Fanuc TP program (LS listing): kj_block_3.ls

/PROG  kj_block_3
/ATTR
COMMENT	= "19-04-11 14:31:32";
PROG_SIZE	= 0;
DEFAULT_GROUP	= 1, *, *, *, *;
/APPL
    ARC Welding Equipment: 1, *, *, *, *;
/MN
   1:  CALL HOME_ALL;
   1:  UFRAME_NUM = 1;
   1:  UTOOL_NUM = 3;
   1:  COL GUARD ADJUST 150;
   1:  MESSAGE[Teach Startpoint in PR90];
   1:  MESSAGE[Weld speed R100 in mm/sec];
   1:  MESSAGE[Retraction +Z in R101 in mm];
   1:  MESSAGE[Retraction speed in R102 in %];
   1:  !- Layer/Ebene 1;
   1:  PR[91] = PR[90];
   1:  PR[91,1] = PR[90,1] + 59.254;
   1:  PR[91,2] = PR[90,2] + 0.794;
   1:  PR[91,3] = PR[90,3] + 1.000;
   1:  PR[92] = PR[91];
   1:  PR[92,3] = PR[92,3] + R[101];
   1:J PR[92] R[102]% CNT100;
   1:L PR[91] 100mm/sec FINE RampTo R[100];
   1:  WAIT   2.00(sec);
   1:  CALL LASER_DRAHT_START;
   1:  PR[91,2] = PR[90,2] + 9.294;
   1:L PR[91] R[100]mm/sec CNT100;
   1:  PR[91,1] = PR[90,1] + 0.754;
   1:L PR[91] R[100]mm/sec CNT100;
   1:  PR[91,2] = PR[90,2] + 0.794;
   1:L PR[91] R[100]mm/sec CNT100;
   1:  PR[91,1] = PR[90,1] + 59.254;
   1:L PR[91] R[100]mm/sec CNT100TB   .50sec,CALL END_PUD;
   1:  WAIT    .50(sec);
   1:  DO[117:Laser Start]=OFF;
   1:  WAIT   10.00(sec);
   1:  PR[92] = PR[91];
   1:  PR[92,3] = PR[92,3] + R[101];
   1:J PR[92] R[102]% CNT100;
   1:  PR[91,1] = PR[90,1] + 56.803;
   1:  PR[91,2] = PR[90,2] + 2.144;
   1:  PR[92] = PR[91];
   1:  PR[92,3] = PR[92,3] + R[101];
   1:J PR[92] R[102]% CNT100;
   1:L PR[91] 100mm/sec FINE RampTo R[100];
   1:  WAIT   2.00(sec);
   1:  CALL LASER_DRAHT_START;
   1:  PR[91,1] = PR[90,1] + 57.904;
   1:  PR[91,2] = PR[90,2] + 3.246;
   1:L PR[91] R[100]mm/sec CNT100;
   1:  PR[91,2] = PR[90,2] + 5.367;
   1:L PR[91] R[100]mm/sec CNT100;
   1:  PR[91,1] = PR[90,1] + 54.681;
   1:  PR[91,2] = PR[90,2] + 2.144;
   1:L PR[91] R[100]mm/sec CNT100;
   1:  PR[91,1] = PR[90,1] + 52.560;
   1:L PR[91] R[100]mm/sec CNT100;
   1:  PR[91,1] = PR[90,1] + 57.904;
   1:  PR[91,2] = PR[90,2] + 7.489;
   1:L PR[91] R[100]mm/sec CNT100;
   1:  PR[91,2] = PR[90,2] + 7.944;
   1:L PR[91] R[100]mm/sec CNT100;
   1:  PR[91,1] = PR[90,1] + 56.239;
   1:L PR[91] R[100]mm/sec CNT100;
   1:  PR[91,1] = PR[90,1] + 50.439;
   1:  PR[91,2] = PR[90,2] + 2.144;
   1:L PR[91] R[100]mm/sec CNT100;
   1:  PR[91,1] = PR[90,1] + 48.317;
   1:L PR[91] R[100]mm/sec CNT100;
   1:  PR[91,1] = PR[90,1] + 54.117;
   1:  PR[91,2] = PR[90,2] + 7.944;
   1:L PR[91] R[100]mm/sec CNT100;
   1:  PR[91,1] = PR[90,1] + 51.996;
   1:L PR[91] R[100]mm/sec CNT100;
   1:  PR[91,1] = PR[90,1] + 46.196;
   1:  PR[91,2] = PR[90,2] + 2.144;
   1:L PR[91] R[100]mm/sec CNT100;
   1:  PR[91,1] = PR[90,1] + 44.075;
   1:L PR[91] R[100]mm/sec CNT100;
   1:  PR[91,1] = PR[90,1] + 49.875;
   1:  PR[91,2] = PR[90,2] + 7.944;
   1:L PR[91] R[100]mm/sec CNT100;
   1:  PR[91,1] = PR[90,1] + 47.753;
   1:L PR[91] R[100]mm/sec CNT100;
   1:  PR[91,1] = PR[90,1] + 41.953;
   1:  PR[91,2] = PR[90,2] + 2.144;
   1:L PR[91] R[100]mm/sec CNT100;
   1:  PR[91,1] = PR[90,1] + 39.832;
   1:L PR[91] R[100]mm/sec CNT100;
   1:  PR[91,1] = PR[90,1] + 45.632;
   1:  PR[91,2] = PR[90,2] + 7.944;
   1:L PR[91] R[100]mm/sec CNT100;
   1:  PR[91,1] = PR[90,1] + 43.511;
   1:L PR[91] R[100]mm/sec CNT100;
   1:  PR[91,1] = PR[90,1] + 37.711;
   1:  PR[91,2] = PR[90,2] + 2.144;
   1:L PR[91] R[100]mm/sec CNT100;
   1:  PR[91,1] = PR[90,1] + 35.589;
   1:L PR[91] R[100]mm/sec CNT100;
   1:  PR[91,1] = PR[90,1] + 41.389;
   1:  PR[91,2] = PR[90,2] + 7.944;
   1:L PR[91] R[100]mm/sec CNT100;
   1:  PR[91,1] = PR[90,1] + 39.268;
   1:L PR[91] R[100]mm/sec CNT100;
   1:  PR[91,1] = PR[90,1] + 33.468;
   1:  PR[91,2] = PR[90,2] + 2.144;
   1:L PR[91] R[100]mm/sec CNT100;
   1:  PR[91,1] = PR[90,1] + 31.347;
   1:L PR[91] R[100]mm/sec CNT100;
   1:  PR[91,1] = PR[90,1] + 37.147;
   1:  PR[91,2] = PR[90,2] + 7.944;
   1:L PR[91] R[100]mm/sec CNT100;
   1:  PR[91,1] = PR[90,1] + 35.025;
   1:L PR[91] R[100]mm/sec CNT100;
   1:  PR[91,1] = PR[90,1] + 29.225;
   1:  PR[91,2] = PR[90,2] + 2.144;
   1:L PR[91] R[100]mm/sec CNT100;
   1:  PR[91,1] = PR[90,1] + 27.104;
   1:L PR[91] R[100]mm/sec CNT100;
   1:  PR[91,1] = PR[90,1] + 32.904;
   1:  PR[91,2] = PR[90,2] + 7.944;
   1:L PR[91] R[100]mm/sec CNT100;
   1:  PR[91,1] = PR[90,1] + 30.783;
   1:L PR[91] R[100]mm/sec CNT100;
   1:  PR[91,1] = PR[90,1] + 24.983;
   1:  PR[91,2] = PR[90,2] + 2.144;
   1:L PR[91] R[100]mm/sec CNT100;
   1:  PR[91,1] = PR[90,1] + 22.862;
   1:L PR[91] R[100]mm/sec CNT100;
   1:  PR[91,1] = PR[90,1] + 28.662;
   1:  PR[91,2] = PR[90,2] + 7.944;
   1:L PR[91] R[100]mm/sec CNT100;
   1:  PR[91,1] = PR[90,1] + 26.540;
   1:L PR[91] R[100]mm/sec CNT100;
   1:  PR[91,1] = PR[90,1] + 20.740;
   1:  PR[91,2] = PR[90,2] + 2.144;
   1:L PR[91] R[100]mm/sec CNT100;
   1:  PR[91,1] = PR[90,1] + 18.619;
   1:L PR[91] R[100]mm/sec CNT100;
   1:  PR[91,1] = PR[90,1] + 24.419;
   1:  PR[91,2] = PR[90,2] + 7.944;
   1:L PR[91] R[100]mm/sec CNT100;
   1:  PR[91,1] = PR[90,1] + 22.298;
   1:L PR[91] R[100]mm/sec CNT100;
   1:  PR[91,1] = PR[90,1] + 16.498;
   1:  PR[91,2] = PR[90,2] + 2.144;
   1:L PR[91] R[100]mm/sec CNT100;
   1:  PR[91,1] = PR[90,1] + 14.376;
   1:L PR[91] R[100]mm/sec CNT100;
   1:  PR[91,1] = PR[90,1] + 20.176;
   1:  PR[91,2] = PR[90,2] + 7.944;
   1:L PR[91] R[100]mm/sec CNT100;
   1:  PR[91,1] = PR[90,1] + 18.055;
   1:L PR[91] R[100]mm/sec CNT100;
   1:  PR[91,1] = PR[90,1] + 12.255;
   1:  PR[91,2] = PR[90,2] + 2.144;
   1:L PR[91] R[100]mm/sec CNT100;
   1:  PR[91,1] = PR[90,1] + 10.134;
   1:L PR[91] R[100]mm/sec CNT100;
   1:  PR[91,1] = PR[90,1] + 15.934;
   1:  PR[91,2] = PR[90,2] + 7.944;
   1:L PR[91] R[100]mm/sec CNT100;
   1:  PR[91,1] = PR[90,1] + 13.812;
   1:L PR[91] R[100]mm/sec CNT100;
   1:  PR[91,1] = PR[90,1] + 8.012;
   1:  PR[91,2] = PR[90,2] + 2.144;
   1:L PR[91] R[100]mm/sec CNT100;
   1:  PR[91,1] = PR[90,1] + 5.891;
   1:L PR[91] R[100]mm/sec CNT100;
   1:  PR[91,1] = PR[90,1] + 11.691;
   1:  PR[91,2] = PR[90,2] + 7.944;
   1:L PR[91] R[100]mm/sec CNT100;
   1:  PR[91,1] = PR[90,1] + 9.570;
   1:L PR[91] R[100]mm/sec CNT100;
   1:  PR[91,1] = PR[90,1] + 3.770;
   1:  PR[91,2] = PR[90,2] + 2.144;
   1:L PR[91] R[100]mm/sec CNT100;
   1:  PR[91,1] = PR[90,1] + 2.104;
   1:L PR[91] R[100]mm/sec CNT100;
   1:  PR[91,2] = PR[90,2] + 2.600;
   1:L PR[91] R[100]mm/sec CNT100;
   1:  PR[91,1] = PR[90,1] + 7.448;
   1:  PR[91,2] = PR[90,2] + 7.944;
   1:L PR[91] R[100]mm/sec CNT100;
   1:  PR[91,1] = PR[90,1] + 5.327;
   1:L PR[91] R[100]mm/sec CNT100;
   1:  PR[91,1] = PR[90,1] + 2.104;
   1:  PR[91,2] = PR[90,2] + 4.722;
   1:L PR[91] R[100]mm/sec CNT100;
   1:  PR[91,2] = PR[90,2] + 6.843;
   1:L PR[91] R[100]mm/sec CNT100;
   1:  PR[91,1] = PR[90,1] + 3.206;
   1:  PR[91,2] = PR[90,2] + 7.944;
   1:L PR[91] R[100]mm/sec CNT100TB   .50sec,CALL END_PUD;
   1:  WAIT    .50(sec);
   1:  DO[117:Laser Start]=OFF;
   1:  WAIT   10.00(sec);
   1:  PR[92] = PR[91];
   1:  PR[92,3] = PR[92,3] + R[101];
   1:J PR[92] R[102]% CNT100;
   1:  !- Layer/Ebene 2;
   1:  PR[91] = PR[90];
   1:  PR[91,1] = PR[90,1] + 59.254;
   1:  PR[91,2] = PR[90,2] + 9.294;
   1:  PR[91,3] = PR[90,3] + 2.000;
   1:  PR[92] = PR[91];
   1:  PR[92,3] = PR[92,3] + R[101];
   1:J PR[92] R[102]% CNT100;
   1:L PR[91] 100mm/sec FINE RampTo R[100];
   1:  WAIT   2.00(sec);
   1:  CALL LASER_DRAHT_START;
   1:  PR[91,1] = PR[90,1] + 0.754;
   1:L PR[91] R[100]mm/sec CNT100;
   1:  PR[91,2] = PR[90,2] + 0.794;
   1:L PR[91] R[100]mm/sec CNT100;
   1:  PR[91,1] = PR[90,1] + 59.254;
   1:L PR[91] R[100]mm/sec CNT100;
   1:  PR[91,2] = PR[90,2] + 9.294;
   1:L PR[91] R[100]mm/sec CNT100TB   .50sec,CALL END_PUD;
   1:  WAIT    .50(sec);
   1:  DO[117:Laser Start]=OFF;
   1:  WAIT   10.00(sec);
   1:  PR[92] = PR[91];
   1:  PR[92,3] = PR[92,3] + R[101];
   1:J PR[92] R[102]% CNT100;
   1:  PR[91,1] = PR[90,1] + 57.904;
   1:  PR[91,2] = PR[90,2] + 6.843;
   1:  PR[92] = PR[91];
   1:  PR[92,3] = PR[92,3] + R[101];
   1:J PR[92] R[102]% CNT100;
   1:L PR[91] 100mm/sec FINE RampTo R[100];
   1:  WAIT   2.00(sec);
   1:  CALL LASER_DRAHT_START;
   1:  PR[91,1] = PR[90,1] + 56.803;
   1:  PR[91,2] = PR[90,2] + 7.944;
   1:L PR[91] R[100]mm/sec CNT100;
   1:  PR[91,1] = PR[90,1] + 54.681;
   1:L PR[91] R[100]mm/sec CNT100;
   1:  PR[91,1] = PR[90,1] + 57.904;
   1:  PR[91,2] = PR[90,2] + 4.722;
   1:L PR[91] R[100]mm/sec CNT100;
   1:  PR[91,2] = PR[90,2] + 2.600;
   1:L PR[91] R[100]mm/sec CNT100;
   1:  PR[91,1] = PR[90,1] + 52.560;
   1:  PR[91,2] = PR[90,2] + 7.944;
   1:L PR[91] R[100]mm/sec CNT100;
   1:  PR[91,1] = PR[90,1] + 50.439;
   1:L PR[91] R[100]mm/sec CNT100;
   1:  PR[91,1] = PR[90,1] + 56.239;
   1:  PR[91,2] = PR[90,2] + 2.144;
   1:L PR[91] R[100]mm/sec CNT100;
   1:  PR[91,1] = PR[90,1] + 54.117;
   1:L PR[91] R[100]mm/sec CNT100;
   1:  PR[91,1] = PR[90,1] + 48.317;
   1:  PR[91,2] = PR[90,2] + 7.944;
   1:L PR[91] R[100]mm/sec CNT100;
   1:  PR[91,1] = PR[90,1] + 46.196;
   1:L PR[91] R[100]mm/sec CNT100;
   1:  PR[91,1] = PR[90,1] + 51.996;
   1:  PR[91,2] = PR[90,2] + 2.144;
   1:L PR[91] R[100]mm/sec CNT100;
   1:  PR[91,1] = PR[90,1] + 49.875;
   1:L PR[91] R[100]mm/sec CNT100;
   1:  PR[91,1] = PR[90,1] + 44.075;
   1:  PR[91,2] = PR[90,2] + 7.944;
   1:L PR[91] R[100]mm/sec CNT100;
   1:  PR[91,1] = PR[90,1] + 41.953;
   1:L PR[91] R[100]mm/sec CNT100;
   1:  PR[91,1] = PR[90,1] + 47.753;
   1:  PR[91,2] = PR[90,2] + 2.144;
   1:L PR[91] R[100]mm/sec CNT100;
   1:  PR[91,1] = PR[90,1] + 45.632;
   1:L PR[91] R[100]mm/sec CNT100;
   1:  PR[91,1] = PR[90,1] + 39.832;
   1:  PR[91,2] = PR[90,2] + 7.944;
   1:L PR[91] R[100]mm/sec CNT100;
   1:  PR[91,1] = PR[90,1] + 37.711;
   1:L PR[91] R[100]mm/sec CNT100;
   1:  PR[91,1] = PR[90,1] + 43.511;
   1:  PR[91,2] = PR[90,2] + 2.144;
   1:L PR[91] R[100]mm/sec CNT100;
   1:  PR[91,1] = PR[90,1] + 41.389;
   1:L PR[91] R[100]mm/sec CNT100;
   1:  PR[91,1] = PR[90,1] + 35.589;
   1:  PR[91,2] = PR[90,2] + 7.944;
   1:L PR[91] R[100]mm/sec CNT100;
   1:  PR[91,1] = PR[90,1] + 33.468;
   1:L PR[91] R[100]mm/sec CNT100;
   1:  PR[91,1] = PR[90,1] + 39.268;
   1:  PR[91,2] = PR[90,2] + 2.144;
   1:L PR[91] R[100]mm/sec CNT100;
   1:  PR[91,1] = PR[90,1] + 37.147;
   1:L PR[91] R[100]mm/sec CNT100;
   1:  PR[91,1] = PR[90,1] + 31.347;
   1:  PR[91,2] = PR[90,2] + 7.944;
   1:L PR[91] R[100]mm/sec CNT100;
   1:  PR[91,1] = PR[90,1] + 29.226;
   1:L PR[91] R[100]mm/sec CNT100;
   1:  PR[91,1] = PR[90,1] + 35.026;
   1:  PR[91,2] = PR[90,2] + 2.144;
   1:L PR[91] R[100]mm/sec CNT100;
   1:  PR[91,1] = PR[90,1] + 32.904;
   1:L PR[91] R[100]mm/sec CNT100;
   1:  PR[91,1] = PR[90,1] + 27.104;
   1:  PR[91,2] = PR[90,2] + 7.944;
   1:L PR[91] R[100]mm/sec CNT100;
   1:  PR[91,1] = PR[90,1] + 24.983;
   1:L PR[91] R[100]mm/sec CNT100;
   1:  PR[91,1] = PR[90,1] + 30.783;
   1:  PR[91,2] = PR[90,2] + 2.144;
   1:L PR[91] R[100]mm/sec CNT100;
   1:  PR[91,1] = PR[90,1] + 28.662;
   1:L PR[91] R[100]mm/sec CNT100;
   1:  PR[91,1] = PR[90,1] + 22.862;
   1:  PR[91,2] = PR[90,2] + 7.944;
   1:L PR[91] R[100]mm/sec CNT100;
   1:  PR[91,1] = PR[90,1] + 20.740;
   1:L PR[91] R[100]mm/sec CNT100;
   1:  PR[91,1] = PR[90,1] + 26.540;
   1:  PR[91,2] = PR[90,2] + 2.144;
   1:L PR[91] R[100]mm/sec CNT100;
   1:  PR[91,1] = PR[90,1] + 24.419;
   1:L PR[91] R[100]mm/sec CNT100;
   1:  PR[91,1] = PR[90,1] + 18.619;
   1:  PR[91,2] = PR[90,2] + 7.944;
   1:L PR[91] R[100]mm/sec CNT100;
   1:  PR[91,1] = PR[90,1] + 16.498;
   1:L PR[91] R[100]mm/sec CNT100;
   1:  PR[91,1] = PR[90,1] + 22.298;
   1:  PR[91,2] = PR[90,2] + 2.144;
   1:L PR[91] R[100]mm/sec CNT100;
   1:  PR[91,1] = PR[90,1] + 20.176;
   1:L PR[91] R[100]mm/sec CNT100;
   1:  PR[91,1] = PR[90,1] + 14.376;
   1:  PR[91,2] = PR[90,2] + 7.944;
   1:L PR[91] R[100]mm/sec CNT100;
   1:  PR[91,1] = PR[90,1] + 12.255;
   1:L PR[91] R[100]mm/sec CNT100;
   1:  PR[91,1] = PR[90,1] + 18.055;
   1:  PR[91,2] = PR[90,2] + 2.144;
   1:L PR[91] R[100]mm/sec CNT100;
   1:  PR[91,1] = PR[90,1] + 15.934;
   1:L PR[91] R[100]mm/sec CNT100;
   1:  PR[91,1] = PR[90,1] + 10.134;
   1:  PR[91,2] = PR[90,2] + 7.944;
   1:L PR[91] R[100]mm/sec CNT100;
   1:  PR[91,1] = PR[90,1] + 8.012;
   1:L PR[91] R[100]mm/sec CNT100;
   1:  PR[91,1] = PR[90,1] + 13.812;
   1:  PR[91,2] = PR[90,2] + 2.144;
   1:L PR[91] R[100]mm/sec CNT100;
   1:  PR[91,1] = PR[90,1] + 11.691;
   1:L PR[91] R[100]mm/sec CNT100;
   1:  PR[91,1] = PR[90,1] + 5.891;
   1:  PR[91,2] = PR[90,2] + 7.944;
   1:L PR[91] R[100]mm/sec CNT100;
   1:  PR[91,1] = PR[90,1] + 3.770;
   1:L PR[91] R[100]mm/sec CNT100;
   1:  PR[91,1] = PR[90,1] + 9.570;
   1:  PR[91,2] = PR[90,2] + 2.144;
   1:L PR[91] R[100]mm/sec CNT100;
   1:  PR[91,1] = PR[90,1] + 7.448;
   1:L PR[91] R[100]mm/sec CNT100;
   1:  PR[91,1] = PR[90,1] + 2.104;
   1:  PR[91,2] = PR[90,2] + 7.489;
   1:L PR[91] R[100]mm/sec CNT100;
   1:  PR[91,2] = PR[90,2] + 5.367;
   1:L PR[91] R[100]mm/sec CNT100;
   1:  PR[91,1] = PR[90,1] + 5.327;
   1:  PR[91,2] = PR[90,2] + 2.144;
   1:L PR[91] R[100]mm/sec CNT100;
   1:  PR[91,1] = PR[90,1] + 3.206;
   1:L PR[91] R[100]mm/sec CNT100;
   1:  PR[91,1] = PR[90,1] + 2.104;
   1:  PR[91,2] = PR[90,2] + 3.246;
   1:L PR[91] R[100]mm/sec CNT100TB   .50sec,CALL END_PUD;
   1:  WAIT    .50(sec);
   1:  DO[117:Laser Start]=OFF;
   1:  WAIT   10.00(sec);
   1:  PR[92] = PR[91];
   1:  PR[92,3] = PR[92,3] + R[101];
   1:J PR[92] R[102]% CNT100;
   1:  !- Layer/Ebene 3;
   1:  PR[91] = PR[90];
   1:  PR[91,1] = PR[90,1] + 59.254;
   1:  PR[91,2] = PR[90,2] + 9.294;
   1:  PR[91,3] = PR[90,3] + 3.000;
   1:  PR[92] = PR[91];
   1:  PR[92,3] = PR[92,3] + R[101];
   1:J PR[92] R[102]% CNT100;
   1:L PR[91] 100mm/sec FINE RampTo R[100];
   1:  WAIT   2.00(sec);
   1:  CALL LASER_DRAHT_START;
   1:  PR[91,1] = PR[90,1] + 0.754;
   1:L PR[91] R[100]mm/sec CNT100;
   1:  PR[91,2] = PR[90,2] + 0.794;
   1:L PR[91] R[100]mm/sec CNT100;
   1:  PR[91,1] = PR[90,1] + 59.254;
   1:L PR[91] R[100]mm/sec CNT100;
   1:  PR[91,2] = PR[90,2] + 9.294;
   1:L PR[91] R[100]mm/sec CNT100TB   .50sec,CALL END_PUD;
   1:  WAIT    .50(sec);
   1:  DO[117:Laser Start]=OFF;
   1:  WAIT   10.00(sec);
   1:  PR[92] = PR[91];
   1:  PR[92,3] = PR[92,3] + R[101];
   1:J PR[92] R[102]% CNT100;
   1:  PR[91,1] = PR[90,1] + 56.803;
   1:  PR[91,2] = PR[90,2] + 2.144;
   1:  PR[92] = PR[91];
   1:  PR[92,3] = PR[92,3] + R[101];
   1:J PR[92] R[102]% CNT100;
   1:L PR[91] 100mm/sec FINE RampTo R[100];
   1:  WAIT   2.00(sec);
   1:  CALL LASER_DRAHT_START;
   1:  PR[91,1] = PR[90,1] + 57.904;
   1:  PR[91,2] = PR[90,2] + 3.246;
   1:L PR[91] R[100]mm/sec CNT100;
   1:  PR[91,2] = PR[90,2] + 5.367;
   1:L PR[91] R[100]mm/sec CNT100;
   1:  PR[91,1] = PR[90,1] + 54.681;
   1:  PR[91,2] = PR[90,2] + 2.144;
   1:L PR[91] R[100]mm/sec CNT100;
   1:  PR[91,1] = PR[90,1] + 52.560;
   1:L PR[91] R[100]mm/sec CNT100;
   1:  PR[91,1] = PR[90,1] + 57.904;
   1:  PR[91,2] = PR[90,2] + 7.489;
   1:L PR[91] R[100]mm/sec CNT100;
   1:  PR[91,2] = PR[90,2] + 7.944;
   1:L PR[91] R[100]mm/sec CNT100;
   1:  PR[91,1] = PR[90,1] + 56.239;
   1:L PR[91] R[100]mm/sec CNT100;
   1:  PR[91,1] = PR[90,1] + 50.439;
   1:  PR[91,2] = PR[90,2] + 2.144;
   1:L PR[91] R[100]mm/sec CNT100;
   1:  PR[91,1] = PR[90,1] + 48.317;
   1:L PR[91] R[100]mm/sec CNT100;
   1:  PR[91,1] = PR[90,1] + 54.117;
   1:  PR[91,2] = PR[90,2] + 7.944;
   1:L PR[91] R[100]mm/sec CNT100;
   1:  PR[91,1] = PR[90,1] + 51.996;
   1:L PR[91] R[100]mm/sec CNT100;
   1:  PR[91,1] = PR[90,1] + 46.196;
   1:  PR[91,2] = PR[90,2] + 2.144;
   1:L PR[91] R[100]mm/sec CNT100;
   1:  PR[91,1] = PR[90,1] + 44.075;
   1:L PR[91] R[100]mm/sec CNT100;
   1:  PR[91,1] = PR[90,1] + 49.875;
   1:  PR[91,2] = PR[90,2] + 7.944;
   1:L PR[91] R[100]mm/sec CNT100;
   1:  PR[91,1] = PR[90,1] + 47.753;
   1:L PR[91] R[100]mm/sec CNT100;
   1:  PR[91,1] = PR[90,1] + 41.953;
   1:  PR[91,2] = PR[90,2] + 2.144;
   1:L PR[91] R[100]mm/sec CNT100;
   1:  PR[91,1] = PR[90,1] + 39.832;
   1:L PR[91] R[100]mm/sec CNT100;
   1:  PR[91,1] = PR[90,1] + 45.632;
   1:  PR[91,2] = PR[90,2] + 7.944;
   1:L PR[91] R[100]mm/sec CNT100;
   1:  PR[91,1] = PR[90,1] + 43.511;
   1:L PR[91] R[100]mm/sec CNT100;
   1:  PR[91,1] = PR[90,1] + 37.711;
   1:  PR[91,2] = PR[90,2] + 2.144;
   1:L PR[91] R[100]mm/sec CNT100;
   1:  PR[91,1] = PR[90,1] + 35.589;
   1:L PR[91] R[100]mm/sec CNT100;
   1:  PR[91,1] = PR[90,1] + 41.389;
   1:  PR[91,2] = PR[90,2] + 7.944;
   1:L PR[91] R[100]mm/sec CNT100;
   1:  PR[91,1] = PR[90,1] + 39.268;
   1:L PR[91] R[100]mm/sec CNT100;
   1:  PR[91,1] = PR[90,1] + 33.468;
   1:  PR[91,2] = PR[90,2] + 2.144;
   1:L PR[91] R[100]mm/sec CNT100;
   1:  PR[91,1] = PR[90,1] + 31.347;
   1:L PR[91] R[100]mm/sec CNT100;
   1:  PR[91,1] = PR[90,1] + 37.147;
   1:  PR[91,2] = PR[90,2] + 7.944;
   1:L PR[91] R[100]mm/sec CNT100;
   1:  PR[91,1] = PR[90,1] + 35.025;
   1:L PR[91] R[100]mm/sec CNT100;
   1:  PR[91,1] = PR[90,1] + 29.225;
   1:  PR[91,2] = PR[90,2] + 2.144;
   1:L PR[91] R[100]mm/sec CNT100;
   1:  PR[91,1] = PR[90,1] + 27.104;
   1:L PR[91] R[100]mm/sec CNT100;
   1:  PR[91,1] = PR[90,1] + 32.904;
   1:  PR[91,2] = PR[90,2] + 7.944;
   1:L PR[91] R[100]mm/sec CNT100;
   1:  PR[91,1] = PR[90,1] + 30.783;
   1:L PR[91] R[100]mm/sec CNT100;
   1:  PR[91,1] = PR[90,1] + 24.983;
   1:  PR[91,2] = PR[90,2] + 2.144;
   1:L PR[91] R[100]mm/sec CNT100;
   1:  PR[91,1] = PR[90,1] + 22.862;
   1:L PR[91] R[100]mm/sec CNT100;
   1:  PR[91,1] = PR[90,1] + 28.662;
   1:  PR[91,2] = PR[90,2] + 7.944;
   1:L PR[91] R[100]mm/sec CNT100;
   1:  PR[91,1] = PR[90,1] + 26.540;
   1:L PR[91] R[100]mm/sec CNT100;
   1:  PR[91,1] = PR[90,1] + 20.740;
   1:  PR[91,2] = PR[90,2] + 2.144;
   1:L PR[91] R[100]mm/sec CNT100;
   1:  PR[91,1] = PR[90,1] + 18.619;
   1:L PR[91] R[100]mm/sec CNT100;
   1:  PR[91,1] = PR[90,1] + 24.419;
   1:  PR[91,2] = PR[90,2] + 7.944;
   1:L PR[91] R[100]mm/sec CNT100;
   1:  PR[91,1] = PR[90,1] + 22.298;
   1:L PR[91] R[100]mm/sec CNT100;
   1:  PR[91,1] = PR[90,1] + 16.498;
   1:  PR[91,2] = PR[90,2] + 2.144;
   1:L PR[91] R[100]mm/sec CNT100;
   1:  PR[91,1] = PR[90,1] + 14.376;
   1:L PR[91] R[100]mm/sec CNT100;
   1:  PR[91,1] = PR[90,1] + 20.176;
   1:  PR[91,2] = PR[90,2] + 7.944;
   1:L PR[91] R[100]mm/sec CNT100;
   1:  PR[91,1] = PR[90,1] + 18.055;
   1:L PR[91] R[100]mm/sec CNT100;
   1:  PR[91,1] = PR[90,1] + 12.255;
   1:  PR[91,2] = PR[90,2] + 2.144;
   1:L PR[91] R[100]mm/sec CNT100;
   1:  PR[91,1] = PR[90,1] + 10.134;
   1:L PR[91] R[100]mm/sec CNT100;
   1:  PR[91,1] = PR[90,1] + 15.934;
   1:  PR[91,2] = PR[90,2] + 7.944;
   1:L PR[91] R[100]mm/sec CNT100;
   1:  PR[91,1] = PR[90,1] + 13.812;
   1:L PR[91] R[100]mm/sec CNT100;
   1:  PR[91,1] = PR[90,1] + 8.012;
   1:  PR[91,2] = PR[90,2] + 2.144;
   1:L PR[91] R[100]mm/sec CNT100;
   1:  PR[91,1] = PR[90,1] + 5.891;
   1:L PR[91] R[100]mm/sec CNT100;
   1:  PR[91,1] = PR[90,1] + 11.691;
   1:  PR[91,2] = PR[90,2] + 7.944;
   1:L PR[91] R[100]mm/sec CNT100;
   1:  PR[91,1] = PR[90,1] + 9.570;
   1:L PR[91] R[100]mm/sec CNT100;
   1:  PR[91,1] = PR[90,1] + 3.770;
   1:  PR[91,2] = PR[90,2] + 2.144;
   1:L PR[91] R[100]mm/sec CNT100;
   1:  PR[91,1] = PR[90,1] + 2.104;
   1:L PR[91] R[100]mm/sec CNT100;
   1:  PR[91,2] = PR[90,2] + 2.600;
   1:L PR[91] R[100]mm/sec CNT100;
   1:  PR[91,1] = PR[90,1] + 7.448;
   1:  PR[91,2] = PR[90,2] + 7.944;
   1:L PR[91] R[100]mm/sec CNT100;
   1:  PR[91,1] = PR[90,1] + 5.327;
   1:L PR[91] R[100]mm/sec CNT100;
   1:  PR[91,1] = PR[90,1] + 2.104;
   1:  PR[91,2] = PR[90,2] + 4.722;
   1:L PR[91] R[100]mm/sec CNT100;
   1:  PR[91,2] = PR[90,2] + 6.843;
   1:L PR[91] R[100]mm/sec CNT100;
   1:  PR[91,1] = PR[90,1] + 3.206;
   1:  PR[91,2] = PR[90,2] + 7.944;
   1:L PR[91] R[100]mm/sec CNT100TB   .50sec,CALL END_PUD;
   1:  WAIT    .50(sec);
   1:  DO[117:Laser Start]=OFF;
   1:  WAIT   10.00(sec);
   1:  PR[92] = PR[91];
   1:  PR[92,3] = PR[92,3] + R[101];
   1:J PR[92] R[102]% CNT100;
   1:  !- Layer/Ebene 4;
   1:  PR[91] = PR[90];
   1:  PR[91,1] = PR[90,1] + 0.754;
   1:  PR[91,2] = PR[90,2] + 0.794;
   1:  PR[91,3] = PR[90,3] + 4.000;
   1:  PR[92] = PR[91];
   1:  PR[92,3] = PR[92,3] + R[101];
   1:J PR[92] R[102]% CNT100;
   1:L PR[91] 100mm/sec FINE RampTo R[100];
   1:  WAIT   2.00(sec);
   1:  CALL LASER_DRAHT_START;
   1:  PR[91,1] = PR[90,1] + 59.254;
   1:L PR[91] R[100]mm/sec CNT100;
   1:  PR[91,2] = PR[90,2] + 9.294;
   1:L PR[91] R[100]mm/sec CNT100;
   1:  PR[91,1] = PR[90,1] + 0.754;
   1:L PR[91] R[100]mm/sec CNT100;
   1:  PR[91,2] = PR[90,2] + 0.794;
   1:L PR[91] R[100]mm/sec CNT100TB   .50sec,CALL END_PUD;
   1:  WAIT    .50(sec);
   1:  DO[117:Laser Start]=OFF;
   1:  WAIT   10.00(sec);
   1:  PR[92] = PR[91];
   1:  PR[92,3] = PR[92,3] + R[101];
   1:J PR[92] R[102]% CNT100;
   1:  PR[91,1] = PR[90,1] + 2.104;
   1:  PR[91,2] = PR[90,2] + 3.246;
   1:  PR[92] = PR[91];
   1:  PR[92,3] = PR[92,3] + R[101];
   1:J PR[92] R[102]% CNT100;
   1:L PR[91] 100mm/sec FINE RampTo R[100];
   1:  WAIT   2.00(sec);
   1:  CALL LASER_DRAHT_START;
   1:  PR[91,1] = PR[90,1] + 3.206;
   1:  PR[91,2] = PR[90,2] + 2.144;
   1:L PR[91] R[100]mm/sec CNT100;
   1:  PR[91,1] = PR[90,1] + 5.327;
   1:L PR[91] R[100]mm/sec CNT100;
   1:  PR[91,1] = PR[90,1] + 2.104;
   1:  PR[91,2] = PR[90,2] + 5.367;
   1:L PR[91] R[100]mm/sec CNT100;
   1:  PR[91,2] = PR[90,2] + 7.489;
   1:L PR[91] R[100]mm/sec CNT100;
   1:  PR[91,1] = PR[90,1] + 7.448;
   1:  PR[91,2] = PR[90,2] + 2.144;
   1:L PR[91] R[100]mm/sec CNT100;
   1:  PR[91,1] = PR[90,1] + 9.570;
   1:L PR[91] R[100]mm/sec CNT100;
   1:  PR[91,1] = PR[90,1] + 3.770;
   1:  PR[91,2] = PR[90,2] + 7.944;
   1:L PR[91] R[100]mm/sec CNT100;
   1:  PR[91,1] = PR[90,1] + 5.891;
   1:L PR[91] R[100]mm/sec CNT100;
   1:  PR[91,1] = PR[90,1] + 11.691;
   1:  PR[91,2] = PR[90,2] + 2.144;
   1:L PR[91] R[100]mm/sec CNT100;
   1:  PR[91,1] = PR[90,1] + 13.812;
   1:L PR[91] R[100]mm/sec CNT100;
   1:  PR[91,1] = PR[90,1] + 8.012;
   1:  PR[91,2] = PR[90,2] + 7.944;
   1:L PR[91] R[100]mm/sec CNT100;
   1:  PR[91,1] = PR[90,1] + 10.134;
   1:L PR[91] R[100]mm/sec CNT100;
   1:  PR[91,1] = PR[90,1] + 15.934;
   1:  PR[91,2] = PR[90,2] + 2.144;
   1:L PR[91] R[100]mm/sec CNT100;
   1:  PR[91,1] = PR[90,1] + 18.055;
   1:L PR[91] R[100]mm/sec CNT100;
   1:  PR[91,1] = PR[90,1] + 12.255;
   1:  PR[91,2] = PR[90,2] + 7.944;
   1:L PR[91] R[100]mm/sec CNT100;
   1:  PR[91,1] = PR[90,1] + 14.376;
   1:L PR[91] R[100]mm/sec CNT100;
   1:  PR[91,1] = PR[90,1] + 20.176;
   1:  PR[91,2] = PR[90,2] + 2.144;
   1:L PR[91] R[100]mm/sec CNT100;
   1:  PR[91,1] = PR[90,1] + 22.298;
   1:L PR[91] R[100]mm/sec CNT100;
   1:  PR[91,1] = PR[90,1] + 16.498;
   1:  PR[91,2] = PR[90,2] + 7.944;
   1:L PR[91] R[100]mm/sec CNT100;
   1:  PR[91,1] = PR[90,1] + 18.619;
   1:L PR[91] R[100]mm/sec CNT100;
   1:  PR[91,1] = PR[90,1] + 24.419;
   1:  PR[91,2] = PR[90,2] + 2.144;
   1:L PR[91] R[100]mm/sec CNT100;
   1:  PR[91,1] = PR[90,1] + 26.540;
   1:L PR[91] R[100]mm/sec CNT100;
   1:  PR[91,1] = PR[90,1] + 20.740;
   1:  PR[91,2] = PR[90,2] + 7.944;
   1:L PR[91] R[100]mm/sec CNT100;
   1:  PR[91,1] = PR[90,1] + 22.862;
   1:L PR[91] R[100]mm/sec CNT100;
   1:  PR[91,1] = PR[90,1] + 28.662;
   1:  PR[91,2] = PR[90,2] + 2.144;
   1:L PR[91] R[100]mm/sec CNT100;
   1:  PR[91,1] = PR[90,1] + 30.783;
   1:L PR[91] R[100]mm/sec CNT100;
   1:  PR[91,1] = PR[90,1] + 24.983;
   1:  PR[91,2] = PR[90,2] + 7.944;
   1:L PR[91] R[100]mm/sec CNT100;
   1:  PR[91,1] = PR[90,1] + 27.104;
   1:L PR[91] R[100]mm/sec CNT100;
   1:  PR[91,1] = PR[90,1] + 32.904;
   1:  PR[91,2] = PR[90,2] + 2.144;
   1:L PR[91] R[100]mm/sec CNT100;
   1:  PR[91,1] = PR[90,1] + 35.026;
   1:L PR[91] R[100]mm/sec CNT100;
   1:  PR[91,1] = PR[90,1] + 29.226;
   1:  PR[91,2] = PR[90,2] + 7.944;
   1:L PR[91] R[100]mm/sec CNT100;
   1:  PR[91,1] = PR[90,1] + 31.347;
   1:L PR[91] R[100]mm/sec CNT100;
   1:  PR[91,1] = PR[90,1] + 37.147;
   1:  PR[91,2] = PR[90,2] + 2.144;
   1:L PR[91] R[100]mm/sec CNT100;
   1:  PR[91,1] = PR[90,1] + 39.268;
   1:L PR[91] R[100]mm/sec CNT100;
   1:  PR[91,1] = PR[90,1] + 33.468;
   1:  PR[91,2] = PR[90,2] + 7.944;
   1:L PR[91] R[100]mm/sec CNT100;
   1:  PR[91,1] = PR[90,1] + 35.589;
   1:L PR[91] R[100]mm/sec CNT100;
   1:  PR[91,1] = PR[90,1] + 41.389;
   1:  PR[91,2] = PR[90,2] + 2.144;
   1:L PR[91] R[100]mm/sec CNT100;
   1:  PR[91,1] = PR[90,1] + 43.511;
   1:L PR[91] R[100]mm/sec CNT100;
   1:  PR[91,1] = PR[90,1] + 37.711;
   1:  PR[91,2] = PR[90,2] + 7.944;
   1:L PR[91] R[100]mm/sec CNT100;
   1:  PR[91,1] = PR[90,1] + 39.832;
   1:L PR[91] R[100]mm/sec CNT100;
   1:  PR[91,1] = PR[90,1] + 45.632;
   1:  PR[91,2] = PR[90,2] + 2.144;
   1:L PR[91] R[100]mm/sec CNT100;
   1:  PR[91,1] = PR[90,1] + 47.753;
   1:L PR[91] R[100]mm/sec CNT100;
   1:  PR[91,1] = PR[90,1] + 41.953;
   1:  PR[91,2] = PR[90,2] + 7.944;
   1:L PR[91] R[100]mm/sec CNT100;
   1:  PR[91,1] = PR[90,1] + 44.075;
   1:L PR[91] R[100]mm/sec CNT100;
   1:  PR[91,1] = PR[90,1] + 49.875;
   1:  PR[91,2] = PR[90,2] + 2.144;
   1:L PR[91] R[100]mm/sec CNT100;
   1:  PR[91,1] = PR[90,1] + 51.996;
   1:L PR[91] R[100]mm/sec CNT100;
   1:  PR[91,1] = PR[90,1] + 46.196;
   1:  PR[91,2] = PR[90,2] + 7.944;
   1:L PR[91] R[100]mm/sec CNT100;
   1:  PR[91,1] = PR[90,1] + 48.317;
   1:L PR[91] R[100]mm/sec CNT100;
   1:  PR[91,1] = PR[90,1] + 54.117;
   1:  PR[91,2] = PR[90,2] + 2.144;
   1:L PR[91] R[100]mm/sec CNT100;
   1:  PR[91,1] = PR[90,1] + 56.239;
   1:L PR[91] R[100]mm/sec CNT100;
   1:  PR[91,1] = PR[90,1] + 50.439;
   1:  PR[91,2] = PR[90,2] + 7.944;
   1:L PR[91] R[100]mm/sec CNT100;
   1:  PR[91,1] = PR[90,1] + 52.560;
   1:L PR[91] R[100]mm/sec CNT100;
   1:  PR[91,1] = PR[90,1] + 57.904;
   1:  PR[91,2] = PR[90,2] + 2.600;
   1:L PR[91] R[100]mm/sec CNT100;
   1:  PR[91,2] = PR[90,2] + 4.722;
   1:L PR[91] R[100]mm/sec CNT100;
   1:  PR[91,1] = PR[90,1] + 54.681;
   1:  PR[91,2] = PR[90,2] + 7.944;
   1:L PR[91] R[100]mm/sec CNT100;
   1:  PR[91,1] = PR[90,1] + 56.803;
   1:L PR[91] R[100]mm/sec CNT100;
   1:  PR[91,1] = PR[90,1] + 57.904;
   1:  PR[91,2] = PR[90,2] + 6.843;
   1:L PR[91] R[100]mm/sec CNT100TB   .50sec,CALL END_PUD;
   1:  WAIT    .50(sec);
   1:  DO[117:Laser Start]=OFF;
   1:  WAIT   10.00(sec);
   1:  PR[92] = PR[91];
   1:  PR[92,3] = PR[92,3] + R[101];
   1:J PR[92] R[102]% CNT100;
   1:  !- Layer/Ebene 5;
   1:  PR[91] = PR[90];
   1:  PR[91,1] = PR[90,1] + 59.254;
   1:  PR[91,2] = PR[90,2] + 9.294;
   1:  PR[91,3] = PR[90,3] + 5.000;
   1:  PR[92] = PR[91];
   1:  PR[92,3] = PR[92,3] + R[101];
   1:J PR[92] R[102]% CNT100;
   1:L PR[91] 100mm/sec FINE RampTo R[100];
   1:  WAIT   2.00(sec);
   1:  CALL LASER_DRAHT_START;
   1:  PR[91,1] = PR[90,1] + 0.754;
   1:L PR[91] R[100]mm/sec CNT100;
   1:  PR[91,2] = PR[90,2] + 0.794;
   1:L PR[91] R[100]mm/sec CNT100;
   1:  PR[91,1] = PR[90,1] + 59.254;
   1:L PR[91] R[100]mm/sec CNT100;
   1:  PR[91,2] = PR[90,2] + 9.294;
   1:L PR[91] R[100]mm/sec CNT100TB   .50sec,CALL END_PUD;
   1:  WAIT    .50(sec);
   1:  DO[117:Laser Start]=OFF;
   1:  WAIT   10.00(sec);
   1:  PR[92] = PR[91];
   1:  PR[92,3] = PR[92,3] + R[101];
   1:J PR[92] R[102]% CNT100;
   1:  PR[91,1] = PR[90,1] + 56.803;
   1:  PR[91,2] = PR[90,2] + 2.144;
   1:  PR[92] = PR[91];
   1:  PR[92,3] = PR[92,3] + R[101];
   1:J PR[92] R[102]% CNT100;
   1:L PR[91] 100mm/sec FINE RampTo R[100];
   1:  WAIT   2.00(sec);
   1:  CALL LASER_DRAHT_START;
   1:  PR[91,1] = PR[90,1] + 57.904;
   1:  PR[91,2] = PR[90,2] + 3.246;
   1:L PR[91] R[100]mm/sec CNT100;
   1:  PR[91,2] = PR[90,2] + 5.367;
   1:L PR[91] R[100]mm/sec CNT100;
   1:  PR[91,1] = PR[90,1] + 54.681;
   1:  PR[91,2] = PR[90,2] + 2.144;
   1:L PR[91] R[100]mm/sec CNT100;
   1:  PR[91,1] = PR[90,1] + 52.560;
   1:L PR[91] R[100]mm/sec CNT100;
   1:  PR[91,1] = PR[90,1] + 57.904;
   1:  PR[91,2] = PR[90,2] + 7.489;
   1:L PR[91] R[100]mm/sec CNT100;
   1:  PR[91,2] = PR[90,2] + 7.944;
   1:L PR[91] R[100]mm/sec CNT100;
   1:  PR[91,1] = PR[90,1] + 56.239;
   1:L PR[91] R[100]mm/sec CNT100;
   1:  PR[91,1] = PR[90,1] + 50.439;
   1:  PR[91,2] = PR[90,2] + 2.144;
   1:L PR[91] R[100]mm/sec CNT100;
   1:  PR[91,1] = PR[90,1] + 48.317;
   1:L PR[91] R[100]mm/sec CNT100;
   1:  PR[91,1] = PR[90,1] + 54.117;
   1:  PR[91,2] = PR[90,2] + 7.944;
   1:L PR[91] R[100]mm/sec CNT100;
   1:  PR[91,1] = PR[90,1] + 51.996;
   1:L PR[91] R[100]mm/sec CNT100;
   1:  PR[91,1] = PR[90,1] + 46.196;
   1:  PR[91,2] = PR[90,2] + 2.144;
   1:L PR[91] R[100]mm/sec CNT100;
   1:  PR[91,1] = PR[90,1] + 44.075;
   1:L PR[91] R[100]mm/sec CNT100;
   1:  PR[91,1] = PR[90,1] + 49.875;
   1:  PR[91,2] = PR[90,2] + 7.944;
   1:L PR[91] R[100]mm/sec CNT100;
   1:  PR[91,1] = PR[90,1] + 47.753;
   1:L PR[91] R[100]mm/sec CNT100;
   1:  PR[91,1] = PR[90,1] + 41.953;
   1:  PR[91,2] = PR[90,2] + 2.144;
   1:L PR[91] R[100]mm/sec CNT100;
   1:  PR[91,1] = PR[90,1] + 39.832;
   1:L PR[91] R[100]mm/sec CNT100;
   1:  PR[91,1] = PR[90,1] + 45.632;
   1:  PR[91,2] = PR[90,2] + 7.944;
   1:L PR[91] R[100]mm/sec CNT100;
   1:  PR[91,1] = PR[90,1] + 43.511;
   1:L PR[91] R[100]mm/sec CNT100;
   1:  PR[91,1] = PR[90,1] + 37.711;
   1:  PR[91,2] = PR[90,2] + 2.144;
   1:L PR[91] R[100]mm/sec CNT100;
   1:  PR[91,1] = PR[90,1] + 35.589;
   1:L PR[91] R[100]mm/sec CNT100;
   1:  PR[91,1] = PR[90,1] + 41.389;
   1:  PR[91,2] = PR[90,2] + 7.944;
   1:L PR[91] R[100]mm/sec CNT100;
   1:  PR[91,1] = PR[90,1] + 39.268;
   1:L PR[91] R[100]mm/sec CNT100;
   1:  PR[91,1] = PR[90,1] + 33.468;
   1:  PR[91,2] = PR[90,2] + 2.144;
   1:L PR[91] R[100]mm/sec CNT100;
   1:  PR[91,1] = PR[90,1] + 31.347;
   1:L PR[91] R[100]mm/sec CNT100;
   1:  PR[91,1] = PR[90,1] + 37.147;
   1:  PR[91,2] = PR[90,2] + 7.944;
   1:L PR[91] R[100]mm/sec CNT100;
   1:  PR[91,1] = PR[90,1] + 35.025;
   1:L PR[91] R[100]mm/sec CNT100;
   1:  PR[91,1] = PR[90,1] + 29.225;
   1:  PR[91,2] = PR[90,2] + 2.144;
   1:L PR[91] R[100]mm/sec CNT100;
   1:  PR[91,1] = PR[90,1] + 27.104;
   1:L PR[91] R[100]mm/sec CNT100;
   1:  PR[91,1] = PR[90,1] + 32.904;
   1:  PR[91,2] = PR[90,2] + 7.944;
   1:L PR[91] R[100]mm/sec CNT100;
   1:  PR[91,1] = PR[90,1] + 30.783;
   1:L PR[91] R[100]mm/sec CNT100;
   1:  PR[91,1] = PR[90,1] + 24.983;
   1:  PR[91,2] = PR[90,2] + 2.144;
   1:L PR[91] R[100]mm/sec CNT100;
   1:  PR[91,1] = PR[90,1] + 22.862;
   1:L PR[91] R[100]mm/sec CNT100;
   1:  PR[91,1] = PR[90,1] + 28.662;
   1:  PR[91,2] = PR[90,2] + 7.944;
   1:L PR[91] R[100]mm/sec CNT100;
   1:  PR[91,1] = PR[90,1] + 26.540;
   1:L PR[91] R[100]mm/sec CNT100;
   1:  PR[91,1] = PR[90,1] + 20.740;
   1:  PR[91,2] = PR[90,2] + 2.144;
   1:L PR[91] R[100]mm/sec CNT100;
   1:  PR[91,1] = PR[90,1] + 18.619;
   1:L PR[91] R[100]mm/sec CNT100;
   1:  PR[91,1] = PR[90,1] + 24.419;
   1:  PR[91,2] = PR[90,2] + 7.944;
   1:L PR[91] R[100]mm/sec CNT100;
   1:  PR[91,1] = PR[90,1] + 22.298;
   1:L PR[91] R[100]mm/sec CNT100;
   1:  PR[91,1] = PR[90,1] + 16.498;
   1:  PR[91,2] = PR[90,2] + 2.144;
   1:L PR[91] R[100]mm/sec CNT100;
   1:  PR[91,1] = PR[90,1] + 14.376;
   1:L PR[91] R[100]mm/sec CNT100;
   1:  PR[91,1] = PR[90,1] + 20.176;
   1:  PR[91,2] = PR[90,2] + 7.944;
   1:L PR[91] R[100]mm/sec CNT100;
   1:  PR[91,1] = PR[90,1] + 18.055;
   1:L PR[91] R[100]mm/sec CNT100;
   1:  PR[91,1] = PR[90,1] + 12.255;
   1:  PR[91,2] = PR[90,2] + 2.144;
   1:L PR[91] R[100]mm/sec CNT100;
   1:  PR[91,1] = PR[90,1] + 10.134;
   1:L PR[91] R[100]mm/sec CNT100;
   1:  PR[91,1] = PR[90,1] + 15.934;
   1:  PR[91,2] = PR[90,2] + 7.944;
   1:L PR[91] R[100]mm/sec CNT100;
   1:  PR[91,1] = PR[90,1] + 13.812;
   1:L PR[91] R[100]mm/sec CNT100;
   1:  PR[91,1] = PR[90,1] + 8.012;
   1:  PR[91,2] = PR[90,2] + 2.144;
   1:L PR[91] R[100]mm/sec CNT100;
   1:  PR[91,1] = PR[90,1] + 5.891;
   1:L PR[91] R[100]mm/sec CNT100;
   1:  PR[91,1] = PR[90,1] + 11.691;
   1:  PR[91,2] = PR[90,2] + 7.944;
   1:L PR[91] R[100]mm/sec CNT100;
   1:  PR[91,1] = PR[90,1] + 9.570;
   1:L PR[91] R[100]mm/sec CNT100;
   1:  PR[91,1] = PR[90,1] + 3.770;
   1:  PR[91,2] = PR[90,2] + 2.144;
   1:L PR[91] R[100]mm/sec CNT100;
   1:  PR[91,1] = PR[90,1] + 2.104;
   1:L PR[91] R[100]mm/sec CNT100;
   1:  PR[91,2] = PR[90,2] + 2.600;
   1:L PR[91] R[100]mm/sec CNT100;
   1:  PR[91,1] = PR[90,1] + 7.448;
   1:  PR[91,2] = PR[90,2] + 7.944;
   1:L PR[91] R[100]mm/sec CNT100;
   1:  PR[91,1] = PR[90,1] + 5.327;
   1:L PR[91] R[100]mm/sec CNT100;
   1:  PR[91,1] = PR[90,1] + 2.104;
   1:  PR[91,2] = PR[90,2] + 4.722;
   1:L PR[91] R[100]mm/sec CNT100;
   1:  PR[91,2] = PR[90,2] + 6.843;
   1:L PR[91] R[100]mm/sec CNT100;
   1:  PR[91,1] = PR[90,1] + 3.206;
   1:  PR[91,2] = PR[90,2] + 7.944;
   1:L PR[91] R[100]mm/sec CNT100TB   .50sec,CALL END_PUD;
   1:  WAIT    .50(sec);
   1:  DO[117:Laser Start]=OFF;
   1:  WAIT   10.00(sec);
   1:  PR[92] = PR[91];
   1:  PR[92,3] = PR[92,3] + R[101];
   1:J PR[92] R[102]% CNT100;
   1:  !- Layer/Ebene 6;
   1:  PR[91] = PR[90];
   1:  PR[91,1] = PR[90,1] + 0.754;
   1:  PR[91,2] = PR[90,2] + 9.294;
   1:  PR[91,3] = PR[90,3] + 6.000;
   1:  PR[92] = PR[91];
   1:  PR[92,3] = PR[92,3] + R[101];
   1:J PR[92] R[102]% CNT100;
   1:L PR[91] 100mm/sec FINE RampTo R[100];
   1:  WAIT   2.00(sec);
   1:  CALL LASER_DRAHT_START;
   1:  PR[91,2] = PR[90,2] + 0.794;
   1:L PR[91] R[100]mm/sec CNT100;
   1:  PR[91,1] = PR[90,1] + 59.254;
   1:L PR[91] R[100]mm/sec CNT100;
   1:  PR[91,2] = PR[90,2] + 9.294;
   1:L PR[91] R[100]mm/sec CNT100;
   1:  PR[91,1] = PR[90,1] + 0.754;
   1:L PR[91] R[100]mm/sec CNT100TB   .50sec,CALL END_PUD;
   1:  WAIT    .50(sec);
   1:  DO[117:Laser Start]=OFF;
   1:  WAIT   10.00(sec);
   1:  PR[92] = PR[91];
   1:  PR[92,3] = PR[92,3] + R[101];
   1:J PR[92] R[102]% CNT100;
   1:  PR[91,1] = PR[90,1] + 2.104;
   1:  PR[91,2] = PR[90,2] + 3.246;
   1:  PR[92] = PR[91];
   1:  PR[92,3] = PR[92,3] + R[101];
   1:J PR[92] R[102]% CNT100;
   1:L PR[91] 100mm/sec FINE RampTo R[100];
   1:  WAIT   2.00(sec);
   1:  CALL LASER_DRAHT_START;
   1:  PR[91,1] = PR[90,1] + 3.206;
   1:  PR[91,2] = PR[90,2] + 2.144;
   1:L PR[91] R[100]mm/sec CNT100;
   1:  PR[91,1] = PR[90,1] + 5.327;
   1:L PR[91] R[100]mm/sec CNT100;
   1:  PR[91,1] = PR[90,1] + 2.104;
   1:  PR[91,2] = PR[90,2] + 5.367;
   1:L PR[91] R[100]mm/sec CNT100;
   1:  PR[91,2] = PR[90,2] + 7.489;
   1:L PR[91] R[100]mm/sec CNT100;
   1:  PR[91,1] = PR[90,1] + 7.448;
   1:  PR[91,2] = PR[90,2] + 2.144;
   1:L PR[91] R[100]mm/sec CNT100;
   1:  PR[91,1] = PR[90,1] + 9.570;
   1:L PR[91] R[100]mm/sec CNT100;
   1:  PR[91,1] = PR[90,1] + 3.770;
   1:  PR[91,2] = PR[90,2] + 7.944;
   1:L PR[91] R[100]mm/sec CNT100;
   1:  PR[91,1] = PR[90,1] + 5.891;
   1:L PR[91] R[100]mm/sec CNT100;
   1:  PR[91,1] = PR[90,1] + 11.691;
   1:  PR[91,2] = PR[90,2] + 2.144;
   1:L PR[91] R[100]mm/sec CNT100;
   1:  PR[91,1] = PR[90,1] + 13.812;
   1:L PR[91] R[100]mm/sec CNT100;
   1:  PR[91,1] = PR[90,1] + 8.012;
   1:  PR[91,2] = PR[90,2] + 7.944;
   1:L PR[91] R[100]mm/sec CNT100;
   1:  PR[91,1] = PR[90,1] + 10.134;
   1:L PR[91] R[100]mm/sec CNT100;
   1:  PR[91,1] = PR[90,1] + 15.934;
   1:  PR[91,2] = PR[90,2] + 2.144;
   1:L PR[91] R[100]mm/sec CNT100;
   1:  PR[91,1] = PR[90,1] + 18.055;
   1:L PR[91] R[100]mm/sec CNT100;
   1:  PR[91,1] = PR[90,1] + 12.255;
   1:  PR[91,2] = PR[90,2] + 7.944;
   1:L PR[91] R[100]mm/sec CNT100;
   1:  PR[91,1] = PR[90,1] + 14.376;
   1:L PR[91] R[100]mm/sec CNT100;
   1:  PR[91,1] = PR[90,1] + 20.176;
   1:  PR[91,2] = PR[90,2] + 2.144;
   1:L PR[91] R[100]mm/sec CNT100;
   1:  PR[91,1] = PR[90,1] + 22.298;
   1:L PR[91] R[100]mm/sec CNT100;
   1:  PR[91,1] = PR[90,1] + 16.498;
   1:  PR[91,2] = PR[90,2] + 7.944;
   1:L PR[91] R[100]mm/sec CNT100;
   1:  PR[91,1] = PR[90,1] + 18.619;
   1:L PR[91] R[100]mm/sec CNT100;
   1:  PR[91,1] = PR[90,1] + 24.419;
   1:  PR[91,2] = PR[90,2] + 2.144;
   1:L PR[91] R[100]mm/sec CNT100;
   1:  PR[91,1] = PR[90,1] + 26.540;
   1:L PR[91] R[100]mm/sec CNT100;
   1:  PR[91,1] = PR[90,1] + 20.740;
   1:  PR[91,2] = PR[90,2] + 7.944;
   1:L PR[91] R[100]mm/sec CNT100;
   1:  PR[91,1] = PR[90,1] + 22.862;
   1:L PR[91] R[100]mm/sec CNT100;
   1:  PR[91,1] = PR[90,1] + 28.662;
   1:  PR[91,2] = PR[90,2] + 2.144;
   1:L PR[91] R[100]mm/sec CNT100;
   1:  PR[91,1] = PR[90,1] + 30.783;
   1:L PR[91] R[100]mm/sec CNT100;
   1:  PR[91,1] = PR[90,1] + 24.983;
   1:  PR[91,2] = PR[90,2] + 7.944;
   1:L PR[91] R[100]mm/sec CNT100;
   1:  PR[91,1] = PR[90,1] + 27.104;
   1:L PR[91] R[100]mm/sec CNT100;
   1:  PR[91,1] = PR[90,1] + 32.904;
   1:  PR[91,2] = PR[90,2] + 2.144;
   1:L PR[91] R[100]mm/sec CNT100;
   1:  PR[91,1] = PR[90,1] + 35.026;
   1:L PR[91] R[100]mm/sec CNT100;
   1:  PR[91,1] = PR[90,1] + 29.226;
   1:  PR[91,2] = PR[90,2] + 7.944;
   1:L PR[91] R[100]mm/sec CNT100;
   1:  PR[91,1] = PR[90,1] + 31.347;
   1:L PR[91] R[100]mm/sec CNT100;
   1:  PR[91,1] = PR[90,1] + 37.147;
   1:  PR[91,2] = PR[90,2] + 2.144;
   1:L PR[91] R[100]mm/sec CNT100;
   1:  PR[91,1] = PR[90,1] + 39.268;
   1:L PR[91] R[100]mm/sec CNT100;
   1:  PR[91,1] = PR[90,1] + 33.468;
   1:  PR[91,2] = PR[90,2] + 7.944;
   1:L PR[91] R[100]mm/sec CNT100;
   1:  PR[91,1] = PR[90,1] + 35.589;
   1:L PR[91] R[100]mm/sec CNT100;
   1:  PR[91,1] = PR[90,1] + 41.389;
   1:  PR[91,2] = PR[90,2] + 2.144;
   1:L PR[91] R[100]mm/sec CNT100;
   1:  PR[91,1] = PR[90,1] + 43.511;
   1:L PR[91] R[100]mm/sec CNT100;
   1:  PR[91,1] = PR[90,1] + 37.711;
   1:  PR[91,2] = PR[90,2] + 7.944;
   1:L PR[91] R[100]mm/sec CNT100;
   1:  PR[91,1] = PR[90,1] + 39.832;
   1:L PR[91] R[100]mm/sec CNT100;
   1:  PR[91,1] = PR[90,1] + 45.632;
   1:  PR[91,2] = PR[90,2] + 2.144;
   1:L PR[91] R[100]mm/sec CNT100;
   1:  PR[91,1] = PR[90,1] + 47.753;
   1:L PR[91] R[100]mm/sec CNT100;
   1:  PR[91,1] = PR[90,1] + 41.953;
   1:  PR[91,2] = PR[90,2] + 7.944;
   1:L PR[91] R[100]mm/sec CNT100;
   1:  PR[91,1] = PR[90,1] + 44.075;
   1:L PR[91] R[100]mm/sec CNT100;
   1:  PR[91,1] = PR[90,1] + 49.875;
   1:  PR[91,2] = PR[90,2] + 2.144;
   1:L PR[91] R[100]mm/sec CNT100;
   1:  PR[91,1] = PR[90,1] + 51.996;
   1:L PR[91] R[100]mm/sec CNT100;
   1:  PR[91,1] = PR[90,1] + 46.196;
   1:  PR[91,2] = PR[90,2] + 7.944;
   1:L PR[91] R[100]mm/sec CNT100;
   1:  PR[91,1] = PR[90,1] + 48.317;
   1:L PR[91] R[100]mm/sec CNT100;
   1:  PR[91,1] = PR[90,1] + 54.117;
   1:  PR[91,2] = PR[90,2] + 2.144;
   1:L PR[91] R[100]mm/sec CNT100;
   1:  PR[91,1] = PR[90,1] + 56.239;
   1:L PR[91] R[100]mm/sec CNT100;
   1:  PR[91,1] = PR[90,1] + 50.439;
   1:  PR[91,2] = PR[90,2] + 7.944;
   1:L PR[91] R[100]mm/sec CNT100;
   1:  PR[91,1] = PR[90,1] + 52.560;
   1:L PR[91] R[100]mm/sec CNT100;
   1:  PR[91,1] = PR[90,1] + 57.904;
   1:  PR[91,2] = PR[90,2] + 2.600;
   1:L PR[91] R[100]mm/sec CNT100;
   1:  PR[91,2] = PR[90,2] + 4.722;
   1:L PR[91] R[100]mm/sec CNT100;
   1:  PR[91,1] = PR[90,1] + 54.681;
   1:  PR[91,2] = PR[90,2] + 7.944;
   1:L PR[91] R[100]mm/sec CNT100;
   1:  PR[91,1] = PR[90,1] + 56.803;
   1:L PR[91] R[100]mm/sec CNT100;
   1:  PR[91,1] = PR[90,1] + 57.904;
   1:  PR[91,2] = PR[90,2] + 6.843;
   1:L PR[91] R[100]mm/sec CNT100TB   .50sec,CALL END_PUD;
   1:  WAIT    .50(sec);
   1:  DO[117:Laser Start]=OFF;
   1:  WAIT   10.00(sec);
   1:  PR[92] = PR[91];
   1:  PR[92,3] = PR[92,3] + R[101];
   1:J PR[92] R[102]% CNT100;
   1:  !- Layer/Ebene 7;
   1:  PR[91] = PR[90];
   1:  PR[91,1] = PR[90,1] + 59.254;
   1:  PR[91,2] = PR[90,2] + 0.794;
   1:  PR[91,3] = PR[90,3] + 7.000;
   1:  PR[92] = PR[91];
   1:  PR[92,3] = PR[92,3] + R[101];
   1:J PR[92] R[102]% CNT100;
   1:L PR[91] 100mm/sec FINE RampTo R[100];
   1:  WAIT   2.00(sec);
   1:  CALL LASER_DRAHT_START;
   1:  PR[91,2] = PR[90,2] + 9.294;
   1:L PR[91] R[100]mm/sec CNT100;
   1:  PR[91,1] = PR[90,1] + 0.754;
   1:L PR[91] R[100]mm/sec CNT100;
   1:  PR[91,2] = PR[90,2] + 0.794;
   1:L PR[91] R[100]mm/sec CNT100;
   1:  PR[91,1] = PR[90,1] + 59.254;
   1:L PR[91] R[100]mm/sec CNT100TB   .50sec,CALL END_PUD;
   1:  WAIT    .50(sec);
   1:  DO[117:Laser Start]=OFF;
   1:  WAIT   10.00(sec);
   1:  PR[92] = PR[91];
   1:  PR[92,3] = PR[92,3] + R[101];
   1:J PR[92] R[102]% CNT100;
   1:  PR[91,1] = PR[90,1] + 56.803;
   1:  PR[91,2] = PR[90,2] + 2.144;
   1:  PR[92] = PR[91];
   1:  PR[92,3] = PR[92,3] + R[101];
   1:J PR[92] R[102]% CNT100;
   1:L PR[91] 100mm/sec FINE RampTo R[100];
   1:  WAIT   2.00(sec);
   1:  CALL LASER_DRAHT_START;
   1:  PR[91,1] = PR[90,1] + 57.904;
   1:  PR[91,2] = PR[90,2] + 3.246;
   1:L PR[91] R[100]mm/sec CNT100;
   1:  PR[91,2] = PR[90,2] + 5.367;
   1:L PR[91] R[100]mm/sec CNT100;
   1:  PR[91,1] = PR[90,1] + 54.681;
   1:  PR[91,2] = PR[90,2] + 2.144;
   1:L PR[91] R[100]mm/sec CNT100;
   1:  PR[91,1] = PR[90,1] + 52.560;
   1:L PR[91] R[100]mm/sec CNT100;
   1:  PR[91,1] = PR[90,1] + 57.904;
   1:  PR[91,2] = PR[90,2] + 7.489;
   1:L PR[91] R[100]mm/sec CNT100;
   1:  PR[91,2] = PR[90,2] + 7.944;
   1:L PR[91] R[100]mm/sec CNT100;
   1:  PR[91,1] = PR[90,1] + 56.239;
   1:L PR[91] R[100]mm/sec CNT100;
   1:  PR[91,1] = PR[90,1] + 50.439;
   1:  PR[91,2] = PR[90,2] + 2.144;
   1:L PR[91] R[100]mm/sec CNT100;
   1:  PR[91,1] = PR[90,1] + 48.317;
   1:L PR[91] R[100]mm/sec CNT100;
   1:  PR[91,1] = PR[90,1] + 54.117;
   1:  PR[91,2] = PR[90,2] + 7.944;
   1:L PR[91] R[100]mm/sec CNT100;
   1:  PR[91,1] = PR[90,1] + 51.996;
   1:L PR[91] R[100]mm/sec CNT100;
   1:  PR[91,1] = PR[90,1] + 46.196;
   1:  PR[91,2] = PR[90,2] + 2.144;
   1:L PR[91] R[100]mm/sec CNT100;
   1:  PR[91,1] = PR[90,1] + 44.075;
   1:L PR[91] R[100]mm/sec CNT100;
   1:  PR[91,1] = PR[90,1] + 49.875;
   1:  PR[91,2] = PR[90,2] + 7.944;
   1:L PR[91] R[100]mm/sec CNT100;
   1:  PR[91,1] = PR[90,1] + 47.753;
   1:L PR[91] R[100]mm/sec CNT100;
   1:  PR[91,1] = PR[90,1] + 41.953;
   1:  PR[91,2] = PR[90,2] + 2.144;
   1:L PR[91] R[100]mm/sec CNT100;
   1:  PR[91,1] = PR[90,1] + 39.832;
   1:L PR[91] R[100]mm/sec CNT100;
   1:  PR[91,1] = PR[90,1] + 45.632;
   1:  PR[91,2] = PR[90,2] + 7.944;
   1:L PR[91] R[100]mm/sec CNT100;
   1:  PR[91,1] = PR[90,1] + 43.511;
   1:L PR[91] R[100]mm/sec CNT100;
   1:  PR[91,1] = PR[90,1] + 37.711;
   1:  PR[91,2] = PR[90,2] + 2.144;
   1:L PR[91] R[100]mm/sec CNT100;
   1:  PR[91,1] = PR[90,1] + 35.589;
   1:L PR[91] R[100]mm/sec CNT100;
   1:  PR[91,1] = PR[90,1] + 41.389;
   1:  PR[91,2] = PR[90,2] + 7.944;
   1:L PR[91] R[100]mm/sec CNT100;
   1:  PR[91,1] = PR[90,1] + 39.268;
   1:L PR[91] R[100]mm/sec CNT100;
   1:  PR[91,1] = PR[90,1] + 33.468;
   1:  PR[91,2] = PR[90,2] + 2.144;
   1:L PR[91] R[100]mm/sec CNT100;
   1:  PR[91,1] = PR[90,1] + 31.347;
   1:L PR[91] R[100]mm/sec CNT100;
   1:  PR[91,1] = PR[90,1] + 37.147;
   1:  PR[91,2] = PR[90,2] + 7.944;
   1:L PR[91] R[100]mm/sec CNT100;
   1:  PR[91,1] = PR[90,1] + 35.025;
   1:L PR[91] R[100]mm/sec CNT100;
   1:  PR[91,1] = PR[90,1] + 29.225;
   1:  PR[91,2] = PR[90,2] + 2.144;
   1:L PR[91] R[100]mm/sec CNT100;
   1:  PR[91,1] = PR[90,1] + 27.104;
   1:L PR[91] R[100]mm/sec CNT100;
   1:  PR[91,1] = PR[90,1] + 32.904;
   1:  PR[91,2] = PR[90,2] + 7.944;
   1:L PR[91] R[100]mm/sec CNT100;
   1:  PR[91,1] = PR[90,1] + 30.783;
   1:L PR[91] R[100]mm/sec CNT100;
   1:  PR[91,1] = PR[90,1] + 24.983;
   1:  PR[91,2] = PR[90,2] + 2.144;
   1:L PR[91] R[100]mm/sec CNT100;
   1:  PR[91,1] = PR[90,1] + 22.862;
   1:L PR[91] R[100]mm/sec CNT100;
   1:  PR[91,1] = PR[90,1] + 28.662;
   1:  PR[91,2] = PR[90,2] + 7.944;
   1:L PR[91] R[100]mm/sec CNT100;
   1:  PR[91,1] = PR[90,1] + 26.540;
   1:L PR[91] R[100]mm/sec CNT100;
   1:  PR[91,1] = PR[90,1] + 20.740;
   1:  PR[91,2] = PR[90,2] + 2.144;
   1:L PR[91] R[100]mm/sec CNT100;
   1:  PR[91,1] = PR[90,1] + 18.619;
   1:L PR[91] R[100]mm/sec CNT100;
   1:  PR[91,1] = PR[90,1] + 24.419;
   1:  PR[91,2] = PR[90,2] + 7.944;
   1:L PR[91] R[100]mm/sec CNT100;
   1:  PR[91,1] = PR[90,1] + 22.298;
   1:L PR[91] R[100]mm/sec CNT100;
   1:  PR[91,1] = PR[90,1] + 16.498;
   1:  PR[91,2] = PR[90,2] + 2.144;
   1:L PR[91] R[100]mm/sec CNT100;
   1:  PR[91,1] = PR[90,1] + 14.376;
   1:L PR[91] R[100]mm/sec CNT100;
   1:  PR[91,1] = PR[90,1] + 20.176;
   1:  PR[91,2] = PR[90,2] + 7.944;
   1:L PR[91] R[100]mm/sec CNT100;
   1:  PR[91,1] = PR[90,1] + 18.055;
   1:L PR[91] R[100]mm/sec CNT100;
   1:  PR[91,1] = PR[90,1] + 12.255;
   1:  PR[91,2] = PR[90,2] + 2.144;
   1:L PR[91] R[100]mm/sec CNT100;
   1:  PR[91,1] = PR[90,1] + 10.134;
   1:L PR[91] R[100]mm/sec CNT100;
   1:  PR[91,1] = PR[90,1] + 15.934;
   1:  PR[91,2] = PR[90,2] + 7.944;
   1:L PR[91] R[100]mm/sec CNT100;
   1:  PR[91,1] = PR[90,1] + 13.812;
   1:L PR[91] R[100]mm/sec CNT100;
   1:  PR[91,1] = PR[90,1] + 8.012;
   1:  PR[91,2] = PR[90,2] + 2.144;
   1:L PR[91] R[100]mm/sec CNT100;
   1:  PR[91,1] = PR[90,1] + 5.891;
   1:L PR[91] R[100]mm/sec CNT100;
   1:  PR[91,1] = PR[90,1] + 11.691;
   1:  PR[91,2] = PR[90,2] + 7.944;
   1:L PR[91] R[100]mm/sec CNT100;
   1:  PR[91,1] = PR[90,1] + 9.570;
   1:L PR[91] R[100]mm/sec CNT100;
   1:  PR[91,1] = PR[90,1] + 3.770;
   1:  PR[91,2] = PR[90,2] + 2.144;
   1:L PR[91] R[100]mm/sec CNT100;
   1:  PR[91,1] = PR[90,1] + 2.104;
   1:L PR[91] R[100]mm/sec CNT100;
   1:  PR[91,2] = PR[90,2] + 2.600;
   1:L PR[91] R[100]mm/sec CNT100;
   1:  PR[91,1] = PR[90,1] + 7.448;
   1:  PR[91,2] = PR[90,2] + 7.944;
   1:L PR[91] R[100]mm/sec CNT100;
   1:  PR[91,1] = PR[90,1] + 5.327;
   1:L PR[91] R[100]mm/sec CNT100;
   1:  PR[91,1] = PR[90,1] + 2.104;
   1:  PR[91,2] = PR[90,2] + 4.722;
   1:L PR[91] R[100]mm/sec CNT100;
   1:  PR[91,2] = PR[90,2] + 6.843;
   1:L PR[91] R[100]mm/sec CNT100;
   1:  PR[91,1] = PR[90,1] + 3.206;
   1:  PR[91,2] = PR[90,2] + 7.944;
   1:L PR[91] R[100]mm/sec CNT100TB   .50sec,CALL END_PUD;
   1:  WAIT    .50(sec);
   1:  DO[117:Laser Start]=OFF;
   1:  WAIT   10.00(sec);
   1:  PR[92] = PR[91];
   1:  PR[92,3] = PR[92,3] + R[101];
   1:J PR[92] R[102]% CNT100;
   1:  !- Layer/Ebene 8;
   1:  PR[91] = PR[90];
   1:  PR[91,1] = PR[90,1] + 59.254;
   1:  PR[91,2] = PR[90,2] + 0.794;
   1:  PR[91,3] = PR[90,3] + 8.000;
   1:  PR[92] = PR[91];
   1:  PR[92,3] = PR[92,3] + R[101];
   1:J PR[92] R[102]% CNT100;
   1:L PR[91] 100mm/sec FINE RampTo R[100];
   1:  WAIT   2.00(sec);
   1:  CALL LASER_DRAHT_START;
   1:  PR[91,2] = PR[90,2] + 9.294;
   1:L PR[91] R[100]mm/sec CNT100;
   1:  PR[91,1] = PR[90,1] + 0.754;
   1:L PR[91] R[100]mm/sec CNT100;
   1:  PR[91,2] = PR[90,2] + 0.794;
   1:L PR[91] R[100]mm/sec CNT100;
   1:  PR[91,1] = PR[90,1] + 59.254;
   1:L PR[91] R[100]mm/sec CNT100TB   .50sec,CALL END_PUD;
   1:  WAIT    .50(sec);
   1:  DO[117:Laser Start]=OFF;
   1:  WAIT   10.00(sec);
   1:  PR[92] = PR[91];
   1:  PR[92,3] = PR[92,3] + R[101];
   1:J PR[92] R[102]% CNT100;
   1:  PR[91,1] = PR[90,1] + 57.904;
   1:  PR[91,2] = PR[90,2] + 6.843;
   1:  PR[92] = PR[91];
   1:  PR[92,3] = PR[92,3] + R[101];
   1:J PR[92] R[102]% CNT100;
   1:L PR[91] 100mm/sec FINE RampTo R[100];
   1:  WAIT   2.00(sec);
   1:  CALL LASER_DRAHT_START;
   1:  PR[91,1] = PR[90,1] + 56.803;
   1:  PR[91,2] = PR[90,2] + 7.944;
   1:L PR[91] R[100]mm/sec CNT100;
   1:  PR[91,1] = PR[90,1] + 54.681;
   1:L PR[91] R[100]mm/sec CNT100;
   1:  PR[91,1] = PR[90,1] + 57.904;
   1:  PR[91,2] = PR[90,2] + 4.722;
   1:L PR[91] R[100]mm/sec CNT100;
   1:  PR[91,2] = PR[90,2] + 2.600;
   1:L PR[91] R[100]mm/sec CNT100;
   1:  PR[91,1] = PR[90,1] + 52.560;
   1:  PR[91,2] = PR[90,2] + 7.944;
   1:L PR[91] R[100]mm/sec CNT100;
   1:  PR[91,1] = PR[90,1] + 50.439;
   1:L PR[91] R[100]mm/sec CNT100;
   1:  PR[91,1] = PR[90,1] + 56.239;
   1:  PR[91,2] = PR[90,2] + 2.144;
   1:L PR[91] R[100]mm/sec CNT100;
   1:  PR[91,1] = PR[90,1] + 54.117;
   1:L PR[91] R[100]mm/sec CNT100;
   1:  PR[91,1] = PR[90,1] + 48.317;
   1:  PR[91,2] = PR[90,2] + 7.944;
   1:L PR[91] R[100]mm/sec CNT100;
   1:  PR[91,1] = PR[90,1] + 46.196;
   1:L PR[91] R[100]mm/sec CNT100;
   1:  PR[91,1] = PR[90,1] + 51.996;
   1:  PR[91,2] = PR[90,2] + 2.144;
   1:L PR[91] R[100]mm/sec CNT100;
   1:  PR[91,1] = PR[90,1] + 49.875;
   1:L PR[91] R[100]mm/sec CNT100;
   1:  PR[91,1] = PR[90,1] + 44.075;
   1:  PR[91,2] = PR[90,2] + 7.944;
   1:L PR[91] R[100]mm/sec CNT100;
   1:  PR[91,1] = PR[90,1] + 41.953;
   1:L PR[91] R[100]mm/sec CNT100;
   1:  PR[91,1] = PR[90,1] + 47.753;
   1:  PR[91,2] = PR[90,2] + 2.144;
   1:L PR[91] R[100]mm/sec CNT100;
   1:  PR[91,1] = PR[90,1] + 45.632;
   1:L PR[91] R[100]mm/sec CNT100;
   1:  PR[91,1] = PR[90,1] + 39.832;
   1:  PR[91,2] = PR[90,2] + 7.944;
   1:L PR[91] R[100]mm/sec CNT100;
   1:  PR[91,1] = PR[90,1] + 37.711;
   1:L PR[91] R[100]mm/sec CNT100;
   1:  PR[91,1] = PR[90,1] + 43.511;
   1:  PR[91,2] = PR[90,2] + 2.144;
   1:L PR[91] R[100]mm/sec CNT100;
   1:  PR[91,1] = PR[90,1] + 41.389;
   1:L PR[91] R[100]mm/sec CNT100;
   1:  PR[91,1] = PR[90,1] + 35.589;
   1:  PR[91,2] = PR[90,2] + 7.944;
   1:L PR[91] R[100]mm/sec CNT100;
   1:  PR[91,1] = PR[90,1] + 33.468;
   1:L PR[91] R[100]mm/sec CNT100;
   1:  PR[91,1] = PR[90,1] + 39.268;
   1:  PR[91,2] = PR[90,2] + 2.144;
   1:L PR[91] R[100]mm/sec CNT100;
   1:  PR[91,1] = PR[90,1] + 37.147;
   1:L PR[91] R[100]mm/sec CNT100;
   1:  PR[91,1] = PR[90,1] + 31.347;
   1:  PR[91,2] = PR[90,2] + 7.944;
   1:L PR[91] R[100]mm/sec CNT100;
   1:  PR[91,1] = PR[90,1] + 29.226;
   1:L PR[91] R[100]mm/sec CNT100;
   1:  PR[91,1] = PR[90,1] + 35.026;
   1:  PR[91,2] = PR[90,2] + 2.144;
   1:L PR[91] R[100]mm/sec CNT100;
   1:  PR[91,1] = PR[90,1] + 32.904;
   1:L PR[91] R[100]mm/sec CNT100;
   1:  PR[91,1] = PR[90,1] + 27.104;
   1:  PR[91,2] = PR[90,2] + 7.944;
   1:L PR[91] R[100]mm/sec CNT100;
   1:  PR[91,1] = PR[90,1] + 24.983;
   1:L PR[91] R[100]mm/sec CNT100;
   1:  PR[91,1] = PR[90,1] + 30.783;
   1:  PR[91,2] = PR[90,2] + 2.144;
   1:L PR[91] R[100]mm/sec CNT100;
   1:  PR[91,1] = PR[90,1] + 28.662;
   1:L PR[91] R[100]mm/sec CNT100;
   1:  PR[91,1] = PR[90,1] + 22.862;
   1:  PR[91,2] = PR[90,2] + 7.944;
   1:L PR[91] R[100]mm/sec CNT100;
   1:  PR[91,1] = PR[90,1] + 20.740;
   1:L PR[91] R[100]mm/sec CNT100;
   1:  PR[91,1] = PR[90,1] + 26.540;
   1:  PR[91,2] = PR[90,2] + 2.144;
   1:L PR[91] R[100]mm/sec CNT100;
   1:  PR[91,1] = PR[90,1] + 24.419;
   1:L PR[91] R[100]mm/sec CNT100;
   1:  PR[91,1] = PR[90,1] + 18.619;
   1:  PR[91,2] = PR[90,2] + 7.944;
   1:L PR[91] R[100]mm/sec CNT100;
   1:  PR[91,1] = PR[90,1] + 16.498;
   1:L PR[91] R[100]mm/sec CNT100;
   1:  PR[91,1] = PR[90,1] + 22.298;
   1:  PR[91,2] = PR[90,2] + 2.144;
   1:L PR[91] R[100]mm/sec CNT100;
   1:  PR[91,1] = PR[90,1] + 20.176;
   1:L PR[91] R[100]mm/sec CNT100;
   1:  PR[91,1] = PR[90,1] + 14.376;
   1:  PR[91,2] = PR[90,2] + 7.944;
   1:L PR[91] R[100]mm/sec CNT100;
   1:  PR[91,1] = PR[90,1] + 12.255;
   1:L PR[91] R[100]mm/sec CNT100;
   1:  PR[91,1] = PR[90,1] + 18.055;
   1:  PR[91,2] = PR[90,2] + 2.144;
   1:L PR[91] R[100]mm/sec CNT100;
   1:  PR[91,1] = PR[90,1] + 15.934;
   1:L PR[91] R[100]mm/sec CNT100;
   1:  PR[91,1] = PR[90,1] + 10.134;
   1:  PR[91,2] = PR[90,2] + 7.944;
   1:L PR[91] R[100]mm/sec CNT100;
   1:  PR[91,1] = PR[90,1] + 8.012;
   1:L PR[91] R[100]mm/sec CNT100;
   1:  PR[91,1] = PR[90,1] + 13.812;
   1:  PR[91,2] = PR[90,2] + 2.144;
   1:L PR[91] R[100]mm/sec CNT100;
   1:  PR[91,1] = PR[90,1] + 11.691;
   1:L PR[91] R[100]mm/sec CNT100;
   1:  PR[91,1] = PR[90,1] + 5.891;
   1:  PR[91,2] = PR[90,2] + 7.944;
   1:L PR[91] R[100]mm/sec CNT100;
   1:  PR[91,1] = PR[90,1] + 3.770;
   1:L PR[91] R[100]mm/sec CNT100;
   1:  PR[91,1] = PR[90,1] + 9.570;
   1:  PR[91,2] = PR[90,2] + 2.144;
   1:L PR[91] R[100]mm/sec CNT100;
   1:  PR[91,1] = PR[90,1] + 7.448;
   1:L PR[91] R[100]mm/sec CNT100;
   1:  PR[91,1] = PR[90,1] + 2.104;
   1:  PR[91,2] = PR[90,2] + 7.489;
   1:L PR[91] R[100]mm/sec CNT100;
   1:  PR[91,2] = PR[90,2] + 5.367;
   1:L PR[91] R[100]mm/sec CNT100;
   1:  PR[91,1] = PR[90,1] + 5.327;
   1:  PR[91,2] = PR[90,2] + 2.144;
   1:L PR[91] R[100]mm/sec CNT100;
   1:  PR[91,1] = PR[90,1] + 3.206;
   1:L PR[91] R[100]mm/sec CNT100;
   1:  PR[91,1] = PR[90,1] + 2.104;
   1:  PR[91,2] = PR[90,2] + 3.246;
   1:L PR[91] R[100]mm/sec CNT100TB   .50sec,CALL END_PUD;
   1:  WAIT    .50(sec);
   1:  DO[117:Laser Start]=OFF;
   1:  WAIT   10.00(sec);
   1:  PR[92] = PR[91];
   1:  PR[92,3] = PR[92,3] + R[101];
   1:J PR[92] R[102]% CNT100;
   1:  !- Layer/Ebene 9;
   1:  PR[91] = PR[90];
   1:  PR[91,1] = PR[90,1] + 0.754;
   1:  PR[91,2] = PR[90,2] + 0.794;
   1:  PR[91,3] = PR[90,3] + 9.000;
   1:  PR[92] = PR[91];
   1:  PR[92,3] = PR[92,3] + R[101];
   1:J PR[92] R[102]% CNT100;
   1:L PR[91] 100mm/sec FINE RampTo R[100];
   1:  WAIT   2.00(sec);
   1:  CALL LASER_DRAHT_START;
   1:  PR[91,1] = PR[90,1] + 59.254;
   1:L PR[91] R[100]mm/sec CNT100;
   1:  PR[91,2] = PR[90,2] + 9.294;
   1:L PR[91] R[100]mm/sec CNT100;
   1:  PR[91,1] = PR[90,1] + 0.754;
   1:L PR[91] R[100]mm/sec CNT100;
   1:  PR[91,2] = PR[90,2] + 0.794;
   1:L PR[91] R[100]mm/sec CNT100TB   .50sec,CALL END_PUD;
   1:  WAIT    .50(sec);
   1:  DO[117:Laser Start]=OFF;
   1:  WAIT   10.00(sec);
   1:  PR[92] = PR[91];
   1:  PR[92,3] = PR[92,3] + R[101];
   1:J PR[92] R[102]% CNT100;
   1:  PR[91,1] = PR[90,1] + 3.206;
   1:  PR[91,2] = PR[90,2] + 7.944;
   1:  PR[92] = PR[91];
   1:  PR[92,3] = PR[92,3] + R[101];
   1:J PR[92] R[102]% CNT100;
   1:L PR[91] 100mm/sec FINE RampTo R[100];
   1:  WAIT   2.00(sec);
   1:  CALL LASER_DRAHT_START;
   1:  PR[91,1] = PR[90,1] + 2.104;
   1:  PR[91,2] = PR[90,2] + 6.843;
   1:L PR[91] R[100]mm/sec CNT100;
   1:  PR[91,2] = PR[90,2] + 4.722;
   1:L PR[91] R[100]mm/sec CNT100;
   1:  PR[91,1] = PR[90,1] + 5.327;
   1:  PR[91,2] = PR[90,2] + 7.944;
   1:L PR[91] R[100]mm/sec CNT100;
   1:  PR[91,1] = PR[90,1] + 7.448;
   1:L PR[91] R[100]mm/sec CNT100;
   1:  PR[91,1] = PR[90,1] + 2.104;
   1:  PR[91,2] = PR[90,2] + 2.600;
   1:L PR[91] R[100]mm/sec CNT100;
   1:  PR[91,2] = PR[90,2] + 2.144;
   1:L PR[91] R[100]mm/sec CNT100;
   1:  PR[91,1] = PR[90,1] + 3.770;
   1:L PR[91] R[100]mm/sec CNT100;
   1:  PR[91,1] = PR[90,1] + 9.570;
   1:  PR[91,2] = PR[90,2] + 7.944;
   1:L PR[91] R[100]mm/sec CNT100;
   1:  PR[91,1] = PR[90,1] + 11.691;
   1:L PR[91] R[100]mm/sec CNT100;
   1:  PR[91,1] = PR[90,1] + 5.891;
   1:  PR[91,2] = PR[90,2] + 2.144;
   1:L PR[91] R[100]mm/sec CNT100;
   1:  PR[91,1] = PR[90,1] + 8.012;
   1:L PR[91] R[100]mm/sec CNT100;
   1:  PR[91,1] = PR[90,1] + 13.812;
   1:  PR[91,2] = PR[90,2] + 7.944;
   1:L PR[91] R[100]mm/sec CNT100;
   1:  PR[91,1] = PR[90,1] + 15.934;
   1:L PR[91] R[100]mm/sec CNT100;
   1:  PR[91,1] = PR[90,1] + 10.134;
   1:  PR[91,2] = PR[90,2] + 2.144;
   1:L PR[91] R[100]mm/sec CNT100;
   1:  PR[91,1] = PR[90,1] + 12.255;
   1:L PR[91] R[100]mm/sec CNT100;
   1:  PR[91,1] = PR[90,1] + 18.055;
   1:  PR[91,2] = PR[90,2] + 7.944;
   1:L PR[91] R[100]mm/sec CNT100;
   1:  PR[91,1] = PR[90,1] + 20.176;
   1:L PR[91] R[100]mm/sec CNT100;
   1:  PR[91,1] = PR[90,1] + 14.376;
   1:  PR[91,2] = PR[90,2] + 2.144;
   1:L PR[91] R[100]mm/sec CNT100;
   1:  PR[91,1] = PR[90,1] + 16.498;
   1:L PR[91] R[100]mm/sec CNT100;
   1:  PR[91,1] = PR[90,1] + 22.298;
   1:  PR[91,2] = PR[90,2] + 7.944;
   1:L PR[91] R[100]mm/sec CNT100;
   1:  PR[91,1] = PR[90,1] + 24.419;
   1:L PR[91] R[100]mm/sec CNT100;
   1:  PR[91,1] = PR[90,1] + 18.619;
   1:  PR[91,2] = PR[90,2] + 2.144;
   1:L PR[91] R[100]mm/sec CNT100;
   1:  PR[91,1] = PR[90,1] + 20.740;
   1:L PR[91] R[100]mm/sec CNT100;
   1:  PR[91,1] = PR[90,1] + 26.540;
   1:  PR[91,2] = PR[90,2] + 7.944;
   1:L PR[91] R[100]mm/sec CNT100;
   1:  PR[91,1] = PR[90,1] + 28.662;
   1:L PR[91] R[100]mm/sec CNT100;
   1:  PR[91,1] = PR[90,1] + 22.862;
   1:  PR[91,2] = PR[90,2] + 2.144;
   1:L PR[91] R[100]mm/sec CNT100;
   1:  PR[91,1] = PR[90,1] + 24.983;
   1:L PR[91] R[100]mm/sec CNT100;
   1:  PR[91,1] = PR[90,1] + 30.783;
   1:  PR[91,2] = PR[90,2] + 7.944;
   1:L PR[91] R[100]mm/sec CNT100;
   1:  PR[91,1] = PR[90,1] + 32.904;
   1:L PR[91] R[100]mm/sec CNT100;
   1:  PR[91,1] = PR[90,1] + 27.104;
   1:  PR[91,2] = PR[90,2] + 2.144;
   1:L PR[91] R[100]mm/sec CNT100;
   1:  PR[91,1] = PR[90,1] + 29.225;
   1:L PR[91] R[100]mm/sec CNT100;
   1:  PR[91,1] = PR[90,1] + 35.025;
   1:  PR[91,2] = PR[90,2] + 7.944;
   1:L PR[91] R[100]mm/sec CNT100;
   1:  PR[91,1] = PR[90,1] + 37.147;
   1:L PR[91] R[100]mm/sec CNT100;
   1:  PR[91,1] = PR[90,1] + 31.347;
   1:  PR[91,2] = PR[90,2] + 2.144;
   1:L PR[91] R[100]mm/sec CNT100;
   1:  PR[91,1] = PR[90,1] + 33.468;
   1:L PR[91] R[100]mm/sec CNT100;
   1:  PR[91,1] = PR[90,1] + 39.268;
   1:  PR[91,2] = PR[90,2] + 7.944;
   1:L PR[91] R[100]mm/sec CNT100;
   1:  PR[91,1] = PR[90,1] + 41.389;
   1:L PR[91] R[100]mm/sec CNT100;
   1:  PR[91,1] = PR[90,1] + 35.589;
   1:  PR[91,2] = PR[90,2] + 2.144;
   1:L PR[91] R[100]mm/sec CNT100;
   1:  PR[91,1] = PR[90,1] + 37.711;
   1:L PR[91] R[100]mm/sec CNT100;
   1:  PR[91,1] = PR[90,1] + 43.511;
   1:  PR[91,2] = PR[90,2] + 7.944;
   1:L PR[91] R[100]mm/sec CNT100;
   1:  PR[91,1] = PR[90,1] + 45.632;
   1:L PR[91] R[100]mm/sec CNT100;
   1:  PR[91,1] = PR[90,1] + 39.832;
   1:  PR[91,2] = PR[90,2] + 2.144;
   1:L PR[91] R[100]mm/sec CNT100;
   1:  PR[91,1] = PR[90,1] + 41.953;
   1:L PR[91] R[100]mm/sec CNT100;
   1:  PR[91,1] = PR[90,1] + 47.753;
   1:  PR[91,2] = PR[90,2] + 7.944;
   1:L PR[91] R[100]mm/sec CNT100;
   1:  PR[91,1] = PR[90,1] + 49.875;
   1:L PR[91] R[100]mm/sec CNT100;
   1:  PR[91,1] = PR[90,1] + 44.075;
   1:  PR[91,2] = PR[90,2] + 2.144;
   1:L PR[91] R[100]mm/sec CNT100;
   1:  PR[91,1] = PR[90,1] + 46.196;
   1:L PR[91] R[100]mm/sec CNT100;
   1:  PR[91,1] = PR[90,1] + 51.996;
   1:  PR[91,2] = PR[90,2] + 7.944;
   1:L PR[91] R[100]mm/sec CNT100;
   1:  PR[91,1] = PR[90,1] + 54.117;
   1:L PR[91] R[100]mm/sec CNT100;
   1:  PR[91,1] = PR[90,1] + 48.317;
   1:  PR[91,2] = PR[90,2] + 2.144;
   1:L PR[91] R[100]mm/sec CNT100;
   1:  PR[91,1] = PR[90,1] + 50.439;
   1:L PR[91] R[100]mm/sec CNT100;
   1:  PR[91,1] = PR[90,1] + 56.239;
   1:  PR[91,2] = PR[90,2] + 7.944;
   1:L PR[91] R[100]mm/sec CNT100;
   1:  PR[91,1] = PR[90,1] + 57.904;
   1:L PR[91] R[100]mm/sec CNT100;
   1:  PR[91,2] = PR[90,2] + 7.489;
   1:L PR[91] R[100]mm/sec CNT100;
   1:  PR[91,1] = PR[90,1] + 52.560;
   1:  PR[91,2] = PR[90,2] + 2.144;
   1:L PR[91] R[100]mm/sec CNT100;
   1:  PR[91,1] = PR[90,1] + 54.681;
   1:L PR[91] R[100]mm/sec CNT100;
   1:  PR[91,1] = PR[90,1] + 57.904;
   1:  PR[91,2] = PR[90,2] + 5.367;
   1:L PR[91] R[100]mm/sec CNT100;
   1:  PR[91,2] = PR[90,2] + 3.246;
   1:L PR[91] R[100]mm/sec CNT100;
   1:  PR[91,1] = PR[90,1] + 56.803;
   1:  PR[91,2] = PR[90,2] + 2.144;
   1:L PR[91] R[100]mm/sec CNT100TB   .50sec,CALL END_PUD;
   1:  WAIT    .50(sec);
   1:  DO[117:Laser Start]=OFF;
   1:  WAIT   10.00(sec);
   1:  PR[92] = PR[91];
   1:  PR[92,3] = PR[92,3] + R[101];
   1:J PR[92] R[102]% CNT100;
   1:  !- Layer/Ebene 10;
   1:  PR[91] = PR[90];
   1:  PR[91,1] = PR[90,1] + 59.254;
   1:  PR[91,2] = PR[90,2] + 9.294;
   1:  PR[91,3] = PR[90,3] + 10.000;
   1:  PR[92] = PR[91];
   1:  PR[92,3] = PR[92,3] + R[101];
   1:J PR[92] R[102]% CNT100;
   1:L PR[91] 100mm/sec FINE RampTo R[100];
   1:  WAIT   2.00(sec);
   1:  CALL LASER_DRAHT_START;
   1:  PR[91,1] = PR[90,1] + 0.754;
   1:L PR[91] R[100]mm/sec CNT100;
   1:  PR[91,2] = PR[90,2] + 0.794;
   1:L PR[91] R[100]mm/sec CNT100;
   1:  PR[91,1] = PR[90,1] + 59.254;
   1:L PR[91] R[100]mm/sec CNT100;
   1:  PR[91,2] = PR[90,2] + 9.294;
   1:L PR[91] R[100]mm/sec CNT100TB   .50sec,CALL END_PUD;
   1:  WAIT    .50(sec);
   1:  DO[117:Laser Start]=OFF;
   1:  WAIT   10.00(sec);
   1:  PR[92] = PR[91];
   1:  PR[92,3] = PR[92,3] + R[101];
   1:J PR[92] R[102]% CNT100;
   1:  PR[91,1] = PR[90,1] + 57.904;
   1:  PR[91,2] = PR[90,2] + 6.843;
   1:  PR[92] = PR[91];
   1:  PR[92,3] = PR[92,3] + R[101];
   1:J PR[92] R[102]% CNT100;
   1:L PR[91] 100mm/sec FINE RampTo R[100];
   1:  WAIT   2.00(sec);
   1:  CALL LASER_DRAHT_START;
   1:  PR[91,1] = PR[90,1] + 56.803;
   1:  PR[91,2] = PR[90,2] + 7.944;
   1:L PR[91] R[100]mm/sec CNT100;
   1:  PR[91,1] = PR[90,1] + 54.681;
   1:L PR[91] R[100]mm/sec CNT100;
   1:  PR[91,1] = PR[90,1] + 57.904;
   1:  PR[91,2] = PR[90,2] + 4.722;
   1:L PR[91] R[100]mm/sec CNT100;
   1:  PR[91,2] = PR[90,2] + 2.600;
   1:L PR[91] R[100]mm/sec CNT100;
   1:  PR[91,1] = PR[90,1] + 52.560;
   1:  PR[91,2] = PR[90,2] + 7.944;
   1:L PR[91] R[100]mm/sec CNT100;
   1:  PR[91,1] = PR[90,1] + 50.439;
   1:L PR[91] R[100]mm/sec CNT100;
   1:  PR[91,1] = PR[90,1] + 56.239;
   1:  PR[91,2] = PR[90,2] + 2.144;
   1:L PR[91] R[100]mm/sec CNT100;
   1:  PR[91,1] = PR[90,1] + 54.117;
   1:L PR[91] R[100]mm/sec CNT100;
   1:  PR[91,1] = PR[90,1] + 48.317;
   1:  PR[91,2] = PR[90,2] + 7.944;
   1:L PR[91] R[100]mm/sec CNT100;
   1:  PR[91,1] = PR[90,1] + 46.196;
   1:L PR[91] R[100]mm/sec CNT100;
   1:  PR[91,1] = PR[90,1] + 51.996;
   1:  PR[91,2] = PR[90,2] + 2.144;
   1:L PR[91] R[100]mm/sec CNT100;
   1:  PR[91,1] = PR[90,1] + 49.875;
   1:L PR[91] R[100]mm/sec CNT100;
   1:  PR[91,1] = PR[90,1] + 44.075;
   1:  PR[91,2] = PR[90,2] + 7.944;
   1:L PR[91] R[100]mm/sec CNT100;
   1:  PR[91,1] = PR[90,1] + 41.953;
   1:L PR[91] R[100]mm/sec CNT100;
   1:  PR[91,1] = PR[90,1] + 47.753;
   1:  PR[91,2] = PR[90,2] + 2.144;
   1:L PR[91] R[100]mm/sec CNT100;
   1:  PR[91,1] = PR[90,1] + 45.632;
   1:L PR[91] R[100]mm/sec CNT100;
   1:  PR[91,1] = PR[90,1] + 39.832;
   1:  PR[91,2] = PR[90,2] + 7.944;
   1:L PR[91] R[100]mm/sec CNT100;
   1:  PR[91,1] = PR[90,1] + 37.711;
   1:L PR[91] R[100]mm/sec CNT100;
   1:  PR[91,1] = PR[90,1] + 43.511;
   1:  PR[91,2] = PR[90,2] + 2.144;
   1:L PR[91] R[100]mm/sec CNT100;
   1:  PR[91,1] = PR[90,1] + 41.389;
   1:L PR[91] R[100]mm/sec CNT100;
   1:  PR[91,1] = PR[90,1] + 35.589;
   1:  PR[91,2] = PR[90,2] + 7.944;
   1:L PR[91] R[100]mm/sec CNT100;
   1:  PR[91,1] = PR[90,1] + 33.468;
   1:L PR[91] R[100]mm/sec CNT100;
   1:  PR[91,1] = PR[90,1] + 39.268;
   1:  PR[91,2] = PR[90,2] + 2.144;
   1:L PR[91] R[100]mm/sec CNT100;
   1:  PR[91,1] = PR[90,1] + 37.147;
   1:L PR[91] R[100]mm/sec CNT100;
   1:  PR[91,1] = PR[90,1] + 31.347;
   1:  PR[91,2] = PR[90,2] + 7.944;
   1:L PR[91] R[100]mm/sec CNT100;
   1:  PR[91,1] = PR[90,1] + 29.226;
   1:L PR[91] R[100]mm/sec CNT100;
   1:  PR[91,1] = PR[90,1] + 35.026;
   1:  PR[91,2] = PR[90,2] + 2.144;
   1:L PR[91] R[100]mm/sec CNT100;
   1:  PR[91,1] = PR[90,1] + 32.904;
   1:L PR[91] R[100]mm/sec CNT100;
   1:  PR[91,1] = PR[90,1] + 27.104;
   1:  PR[91,2] = PR[90,2] + 7.944;
   1:L PR[91] R[100]mm/sec CNT100;
   1:  PR[91,1] = PR[90,1] + 24.983;
   1:L PR[91] R[100]mm/sec CNT100;
   1:  PR[91,1] = PR[90,1] + 30.783;
   1:  PR[91,2] = PR[90,2] + 2.144;
   1:L PR[91] R[100]mm/sec CNT100;
   1:  PR[91,1] = PR[90,1] + 28.662;
   1:L PR[91] R[100]mm/sec CNT100;
   1:  PR[91,1] = PR[90,1] + 22.862;
   1:  PR[91,2] = PR[90,2] + 7.944;
   1:L PR[91] R[100]mm/sec CNT100;
   1:  PR[91,1] = PR[90,1] + 20.740;
   1:L PR[91] R[100]mm/sec CNT100;
   1:  PR[91,1] = PR[90,1] + 26.540;
   1:  PR[91,2] = PR[90,2] + 2.144;
   1:L PR[91] R[100]mm/sec CNT100;
   1:  PR[91,1] = PR[90,1] + 24.419;
   1:L PR[91] R[100]mm/sec CNT100;
   1:  PR[91,1] = PR[90,1] + 18.619;
   1:  PR[91,2] = PR[90,2] + 7.944;
   1:L PR[91] R[100]mm/sec CNT100;
   1:  PR[91,1] = PR[90,1] + 16.498;
   1:L PR[91] R[100]mm/sec CNT100;
   1:  PR[91,1] = PR[90,1] + 22.298;
   1:  PR[91,2] = PR[90,2] + 2.144;
   1:L PR[91] R[100]mm/sec CNT100;
   1:  PR[91,1] = PR[90,1] + 20.176;
   1:L PR[91] R[100]mm/sec CNT100;
   1:  PR[91,1] = PR[90,1] + 14.376;
   1:  PR[91,2] = PR[90,2] + 7.944;
   1:L PR[91] R[100]mm/sec CNT100;
   1:  PR[91,1] = PR[90,1] + 12.255;
   1:L PR[91] R[100]mm/sec CNT100;
   1:  PR[91,1] = PR[90,1] + 18.055;
   1:  PR[91,2] = PR[90,2] + 2.144;
   1:L PR[91] R[100]mm/sec CNT100;
   1:  PR[91,1] = PR[90,1] + 15.934;
   1:L PR[91] R[100]mm/sec CNT100;
   1:  PR[91,1] = PR[90,1] + 10.134;
   1:  PR[91,2] = PR[90,2] + 7.944;
   1:L PR[91] R[100]mm/sec CNT100;
   1:  PR[91,1] = PR[90,1] + 8.012;
   1:L PR[91] R[100]mm/sec CNT100;
   1:  PR[91,1] = PR[90,1] + 13.812;
   1:  PR[91,2] = PR[90,2] + 2.144;
   1:L PR[91] R[100]mm/sec CNT100;
   1:  PR[91,1] = PR[90,1] + 11.691;
   1:L PR[91] R[100]mm/sec CNT100;
   1:  PR[91,1] = PR[90,1] + 5.891;
   1:  PR[91,2] = PR[90,2] + 7.944;
   1:L PR[91] R[100]mm/sec CNT100;
   1:  PR[91,1] = PR[90,1] + 3.770;
   1:L PR[91] R[100]mm/sec CNT100;
   1:  PR[91,1] = PR[90,1] + 9.570;
   1:  PR[91,2] = PR[90,2] + 2.144;
   1:L PR[91] R[100]mm/sec CNT100;
   1:  PR[91,1] = PR[90,1] + 7.448;
   1:L PR[91] R[100]mm/sec CNT100;
   1:  PR[91,1] = PR[90,1] + 2.104;
   1:  PR[91,2] = PR[90,2] + 7.489;
   1:L PR[91] R[100]mm/sec CNT100;
   1:  PR[91,2] = PR[90,2] + 5.367;
   1:L PR[91] R[100]mm/sec CNT100;
   1:  PR[91,1] = PR[90,1] + 5.327;
   1:  PR[91,2] = PR[90,2] + 2.144;
   1:L PR[91] R[100]mm/sec CNT100;
   1:  PR[91,1] = PR[90,1] + 3.206;
   1:L PR[91] R[100]mm/sec CNT100;
   1:  PR[91,1] = PR[90,1] + 2.104;
   1:  PR[91,2] = PR[90,2] + 3.246;
   1:L PR[91] R[100]mm/sec CNT100 TB   .50sec,CALL END_PUD;
   1:  DO[117:Laser Start]=OFF;
   1:  !Sicherheitspunkt!;
   1:  PR[92] = PR[91];
   1:  PR[92,3] = PR[92,3] + 100;
   1:J PR[92] R[102]% CNT100;
   1:  WAIT   5.00(sec);
   1:  DO[119:Gas]=OFF;
   1:  CALL HOME_ALL;
/POS
/END
